Yaskawa INFORM job: A_ROOF_SIDE_0617_2_PAINT_37.JBI

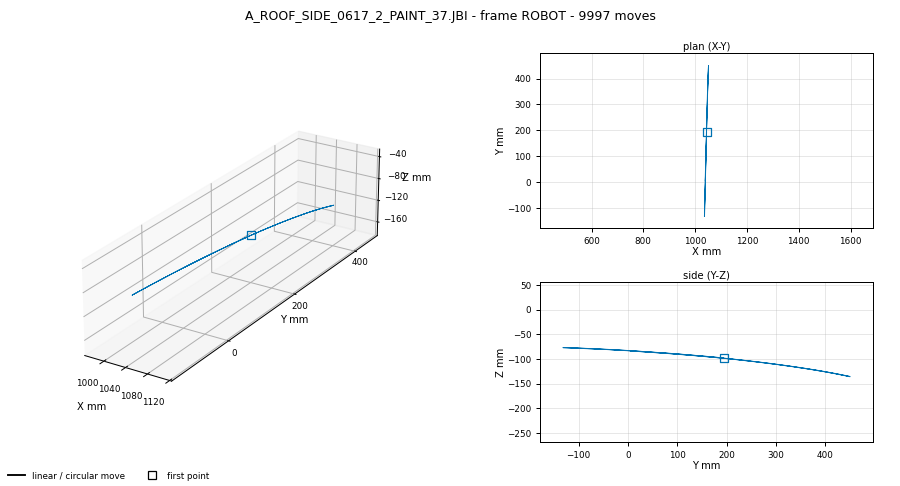
[picture p0: tool path of A_ROOF_SIDE_0617_2_PAINT_37.JBI in frame ROBOT, 9997 of 9997 moves have a stored position in this frame; points joined in program order, loops and branches not executed]
/JOB
//NAME A_ROOF_SIDE_0617_2_PAINT37
//POS
///NPOS 9997,0,0,0,0,0
///TOOL 1
///USER 0
///POSTYPE ROBOT
///RECTAN
///RCONF 1,0,0,0,0,0,0,0,0,0,0,0,0,0,0,0,0,0,0,0,0,0,0,0
C00000=1044.665,193.952,-97.455,170.911,38.372,157.245
C00001=1044.658,193.704,-97.430,170.909,38.370,157.244
C00002=1044.653,193.455,-97.406,170.907,38.368,157.244
C00003=1044.647,193.206,-97.381,170.903,38.367,157.243
C00004=1044.641,192.958,-97.357,170.901,38.365,157.243
C00005=1044.635,192.709,-97.332,170.899,38.364,157.243
C00006=1044.628,192.460,-97.308,170.895,38.362,157.242
C00007=1044.623,192.211,-97.284,170.893,38.360,157.242
C00008=1044.616,191.962,-97.260,170.891,38.359,157.241
C00009=1044.611,191.714,-97.235,170.888,38.357,157.241
C00010=1044.604,191.465,-97.211,170.885,38.355,157.241
C00011=1044.598,191.216,-97.186,170.883,38.353,157.240
C00012=1044.592,190.968,-97.162,170.880,38.352,157.240
C00013=1044.586,190.719,-97.138,170.877,38.350,157.239
C00014=1044.580,190.470,-97.114,170.875,38.348,157.239
C00015=1044.574,190.221,-97.089,170.872,38.347,157.239
C00016=1044.567,189.937,-97.061,170.869,38.345,157.238
C00017=1044.561,189.653,-97.034,170.867,38.342,157.238
C00018=1044.553,189.368,-97.006,170.863,38.341,157.237
C00019=1044.547,189.083,-96.978,170.860,38.339,157.237
C00020=1044.541,188.835,-96.955,170.858,38.337,157.236
C00021=1044.535,188.586,-96.930,170.855,38.336,157.236
C00022=1044.529,188.337,-96.906,170.853,38.334,157.236
C00023=1044.523,188.088,-96.882,170.850,38.332,157.235
C00024=1044.517,187.840,-96.858,170.847,38.330,157.235
C00025=1044.511,187.591,-96.833,170.845,38.329,157.234
C00026=1044.505,187.343,-96.809,170.843,38.327,157.234
C00027=1044.499,187.094,-96.784,170.840,38.325,157.234
C00028=1044.493,186.845,-96.761,170.837,38.323,157.233
C00029=1044.487,186.596,-96.736,170.835,38.322,157.233
C00030=1044.481,186.347,-96.713,170.832,38.320,157.232
C00031=1044.475,186.098,-96.689,170.830,38.319,157.232
C00032=1044.469,185.850,-96.665,170.827,38.317,157.232
C00033=1044.463,185.600,-96.640,170.824,38.315,157.231
C00034=1044.457,185.352,-96.617,170.822,38.313,157.231
C00035=1044.451,185.104,-96.593,170.820,38.312,157.230
C00036=1044.445,184.854,-96.568,170.817,38.310,157.230
C00037=1044.439,184.606,-96.545,170.814,38.308,157.230
C00038=1044.433,184.357,-96.520,170.812,38.307,157.229
C00039=1044.427,184.109,-96.496,170.809,38.305,157.229
C00040=1044.422,183.859,-96.472,170.807,38.304,157.229
C00041=1044.416,183.610,-96.449,170.805,38.302,157.228
C00042=1044.409,183.361,-96.425,170.801,38.300,157.228
C00043=1044.403,183.113,-96.401,170.799,38.299,157.227
C00044=1044.396,182.864,-96.377,170.797,38.297,157.227
C00045=1044.391,182.615,-96.354,170.795,38.296,157.227
C00046=1044.384,182.366,-96.330,170.791,38.294,157.226
C00047=1044.378,182.118,-96.307,170.789,38.293,157.226
C00048=1044.372,181.868,-96.283,170.787,38.291,157.226
C00049=1044.366,181.620,-96.260,170.784,38.290,157.225
C00050=1044.358,181.371,-96.236,170.781,38.289,157.225
C00051=1044.353,181.123,-96.213,170.779,38.287,157.225
C00052=1044.346,180.874,-96.189,170.777,38.286,157.224
C00053=1044.340,180.625,-96.166,170.774,38.284,157.224
C00054=1044.334,180.376,-96.143,170.771,38.283,157.224
C00055=1044.328,180.127,-96.118,170.769,38.281,157.223
C00056=1044.322,179.879,-96.096,170.766,38.279,157.223
C00057=1044.315,179.630,-96.072,170.764,38.278,157.223
C00058=1044.309,179.381,-96.049,170.762,38.276,157.222
C00059=1044.303,179.132,-96.025,170.758,38.275,157.222
C00060=1044.297,178.883,-96.001,170.756,38.274,157.222
C00061=1044.291,178.635,-95.978,170.754,38.272,157.221
C00062=1044.284,178.386,-95.955,170.752,38.271,157.221
C00063=1044.278,178.137,-95.932,170.749,38.270,157.221
C00064=1044.271,177.888,-95.908,170.746,38.268,157.220
C00065=1044.266,177.639,-95.885,170.744,38.266,157.220
C00066=1044.260,177.391,-95.861,170.741,38.265,157.219
C00067=1044.253,177.141,-95.838,170.739,38.263,157.219
C00068=1044.247,176.893,-95.814,170.737,38.262,157.219
C00069=1044.241,176.643,-95.791,170.734,38.260,157.218
C00070=1044.235,176.394,-95.768,170.731,38.259,157.218
C00071=1044.229,176.146,-95.744,170.729,38.257,157.218
C00072=1044.222,175.897,-95.721,170.727,38.256,157.217
C00073=1044.216,175.649,-95.698,170.724,38.255,157.217
C00074=1044.210,175.400,-95.675,170.722,38.253,157.217
C00075=1044.204,175.151,-95.651,170.719,38.252,157.216
C00076=1044.198,174.902,-95.628,170.717,38.251,157.216
C00077=1044.192,174.653,-95.605,170.714,38.249,157.216
C00078=1044.186,174.405,-95.581,170.712,38.248,157.215
C00079=1044.180,174.155,-95.558,170.710,38.246,157.215
C00080=1044.173,173.871,-95.531,170.706,38.244,157.215
C00081=1044.166,173.586,-95.505,170.704,38.242,157.214
C00082=1044.158,173.301,-95.479,170.701,38.241,157.214
C00083=1044.152,173.016,-95.452,170.699,38.239,157.214
C00084=1044.146,172.767,-95.428,170.696,38.238,157.213
C00085=1044.140,172.518,-95.405,170.694,38.237,157.213
C00086=1044.133,172.270,-95.382,170.692,38.235,157.212
C00087=1044.127,172.020,-95.359,170.689,38.234,157.212
C00088=1044.121,171.771,-95.336,170.686,38.232,157.212
C00089=1044.115,171.523,-95.312,170.684,38.231,157.212
C00090=1044.109,171.274,-95.290,170.682,38.229,157.211
C00091=1044.103,171.025,-95.267,170.679,38.228,157.211
C00092=1044.097,170.776,-95.243,170.677,38.226,157.210
C00093=1044.091,170.527,-95.221,170.675,38.224,157.210
C00094=1044.085,170.279,-95.197,170.672,38.223,157.210
C00095=1044.079,170.030,-95.174,170.670,38.221,157.209
C00096=1044.073,169.781,-95.151,170.668,38.220,157.209
C00097=1044.067,169.532,-95.128,170.665,38.219,157.209
C00098=1044.061,169.283,-95.105,170.662,38.217,157.208
C00099=1044.054,169.035,-95.082,170.660,38.216,157.208
C00100=1044.049,168.786,-95.059,170.658,38.214,157.208
C00101=1044.043,168.537,-95.036,170.656,38.213,157.208
C00102=1044.037,168.287,-95.013,170.653,38.212,157.207
C00103=1044.031,168.038,-94.990,170.651,38.210,157.207
C00104=1044.025,167.789,-94.967,170.649,38.209,157.206
C00105=1044.019,167.541,-94.945,170.646,38.207,157.206
C00106=1044.013,167.293,-94.921,170.644,38.206,157.206
C00107=1044.007,167.044,-94.898,170.642,38.205,157.205
C00108=1044.001,166.795,-94.875,170.640,38.203,157.205
C00109=1043.995,166.546,-94.852,170.636,38.202,157.205
C00110=1043.989,166.296,-94.829,170.634,38.200,157.204
C00111=1043.983,166.048,-94.806,170.632,38.199,157.204
C00112=1043.977,165.799,-94.784,170.629,38.197,157.204
C00113=1043.971,165.550,-94.761,170.627,38.196,157.203
C00114=1043.965,165.301,-94.738,170.625,38.194,157.203
C00115=1043.960,165.052,-94.715,170.623,38.193,157.203
C00116=1043.953,164.804,-94.692,170.620,38.191,157.202
C00117=1043.947,164.555,-94.669,170.618,38.190,157.202
C00118=1043.942,164.306,-94.646,170.616,38.188,157.202
C00119=1043.936,164.057,-94.623,170.614,38.187,157.201
C00120=1043.930,163.808,-94.601,170.611,38.185,157.201
C00121=1043.924,163.559,-94.578,170.609,38.184,157.201
C00122=1043.917,163.310,-94.555,170.607,38.182,157.200
C00123=1043.912,163.061,-94.532,170.604,38.181,157.200
C00124=1043.906,162.812,-94.509,170.602,38.179,157.200
C00125=1043.900,162.563,-94.487,170.600,38.178,157.199
C00126=1043.894,162.315,-94.464,170.598,38.177,157.199
C00127=1043.888,162.066,-94.441,170.595,38.175,157.199
C00128=1043.882,161.817,-94.418,170.593,38.174,157.199
C00129=1043.877,161.568,-94.395,170.591,38.172,157.198
C00130=1043.870,161.319,-94.373,170.589,38.171,157.198
C00131=1043.865,161.070,-94.350,170.586,38.170,157.197
C00132=1043.859,160.821,-94.327,170.584,38.168,157.197
C00133=1043.853,160.572,-94.304,170.582,38.167,157.197
C00134=1043.847,160.323,-94.282,170.580,38.165,157.197
C00135=1043.841,160.074,-94.259,170.577,38.164,157.196
C00136=1043.835,159.825,-94.237,170.575,38.162,157.196
C00137=1043.829,159.576,-94.214,170.573,38.161,157.196
C00138=1043.823,159.328,-94.192,170.571,38.160,157.195
C00139=1043.817,159.079,-94.171,170.568,38.158,157.195
C00140=1043.811,158.830,-94.148,170.565,38.157,157.195
C00141=1043.804,158.581,-94.125,170.563,38.156,157.194
C00142=1043.799,158.332,-94.102,170.561,38.155,157.194
C00143=1043.792,158.083,-94.081,170.558,38.153,157.194
C00144=1043.785,157.798,-94.055,170.556,38.152,157.193
C00145=1043.778,157.513,-94.030,170.554,38.150,157.193
C00146=1043.771,157.228,-94.004,170.550,38.149,157.193
C00147=1043.764,156.941,-93.978,170.548,38.147,157.192
C00148=1043.758,156.693,-93.955,170.546,38.146,157.192
C00149=1043.752,156.444,-93.934,170.544,38.145,157.192
C00150=1043.746,156.195,-93.911,170.541,38.143,157.191
C00151=1043.740,155.946,-93.889,170.539,38.142,157.191
C00152=1043.733,155.697,-93.867,170.537,38.141,157.191
C00153=1043.728,155.448,-93.844,170.535,38.140,157.191
C00154=1043.722,155.199,-93.822,170.532,38.138,157.190
C00155=1043.715,154.950,-93.800,170.530,38.137,157.190
C00156=1043.710,154.701,-93.778,170.528,38.136,157.190
C00157=1043.703,154.452,-93.755,170.526,38.135,157.189
C00158=1043.698,154.204,-93.734,170.523,38.133,157.189
C00159=1043.692,153.955,-93.711,170.521,38.132,157.189
C00160=1043.686,153.706,-93.689,170.519,38.130,157.189
C00161=1043.679,153.457,-93.667,170.517,38.129,157.188
C00162=1043.673,153.208,-93.645,170.515,38.128,157.188
C00163=1043.667,152.959,-93.622,170.512,38.126,157.188
C00164=1043.661,152.710,-93.601,170.510,38.125,157.187
C00165=1043.655,152.461,-93.578,170.508,38.124,157.187
C00166=1043.649,152.212,-93.557,170.506,38.123,157.187
C00167=1043.642,151.963,-93.534,170.503,38.122,157.187
C00168=1043.637,151.714,-93.512,170.501,38.121,157.186
C00169=1043.631,151.465,-93.491,170.499,38.119,157.186
C00170=1043.624,151.216,-93.468,170.497,38.118,157.186
C00171=1043.618,150.967,-93.447,170.494,38.116,157.185
C00172=1043.611,150.718,-93.424,170.492,38.115,157.185
C00173=1043.607,150.469,-93.402,170.490,38.114,157.185
C00174=1043.600,150.220,-93.381,170.488,38.112,157.184
C00175=1043.594,149.972,-93.358,170.485,38.111,157.184
C00176=1043.588,149.722,-93.337,170.483,38.110,157.184
C00177=1043.582,149.473,-93.315,170.481,38.109,157.184
C00178=1043.576,149.224,-93.292,170.479,38.108,157.183
C00179=1043.570,148.975,-93.271,170.478,38.107,157.183
C00180=1043.564,148.726,-93.249,170.475,38.105,157.183
C00181=1043.558,148.478,-93.227,170.473,38.104,157.182
C00182=1043.552,148.229,-93.205,170.471,38.102,157.182
C00183=1043.545,147.980,-93.184,170.469,38.101,157.182
C00184=1043.539,147.731,-93.161,170.466,38.100,157.182
C00185=1043.533,147.482,-93.140,170.464,38.099,157.181
C00186=1043.527,147.232,-93.117,170.462,38.098,157.181
C00187=1043.521,146.983,-93.096,170.460,38.097,157.181
C00188=1043.515,146.734,-93.074,170.457,38.095,157.180
C00189=1043.509,146.486,-93.052,170.455,38.094,157.180
C00190=1043.503,146.237,-93.031,170.453,38.092,157.180
C00191=1043.496,145.988,-93.010,170.451,38.091,157.180
C00192=1043.490,145.739,-92.988,170.448,38.090,157.179
C00193=1043.484,145.489,-92.966,170.446,38.089,157.179
C00194=1043.478,145.240,-92.945,170.444,38.088,157.179
C00195=1043.472,144.992,-92.923,170.442,38.087,157.178
C00196=1043.466,144.743,-92.901,170.440,38.086,157.178
C00197=1043.459,144.494,-92.879,170.437,38.084,157.178
C00198=1043.453,144.245,-92.858,170.435,38.083,157.178
C00199=1043.447,143.996,-92.836,170.433,38.082,157.177
C00200=1043.441,143.746,-92.814,170.432,38.081,157.177
C00201=1043.435,143.498,-92.793,170.430,38.080,157.177
C00202=1043.429,143.249,-92.772,170.427,38.078,157.177
C00203=1043.423,142.999,-92.750,170.425,38.077,157.176
C00204=1043.417,142.751,-92.728,170.423,38.076,157.176
C00205=1043.410,142.502,-92.706,170.421,38.074,157.176
C00206=1043.405,142.253,-92.685,170.418,38.073,157.175
C00207=1043.399,142.004,-92.663,170.416,38.072,157.175
C00208=1043.391,141.718,-92.639,170.414,38.071,157.175
C00209=1043.385,141.433,-92.614,170.412,38.070,157.175
C00210=1043.378,141.146,-92.589,170.408,38.068,157.174
C00211=1043.370,140.862,-92.565,170.406,38.067,157.174
C00212=1043.364,140.612,-92.543,170.404,38.066,157.174
C00213=1043.358,140.363,-92.522,170.402,38.064,157.173
C00214=1043.352,140.115,-92.501,170.401,38.063,157.173
C00215=1043.346,139.865,-92.479,170.398,38.062,157.173
C00216=1043.340,139.616,-92.457,170.396,38.060,157.173
C00217=1043.334,139.367,-92.436,170.394,38.059,157.172
C00218=1043.328,139.119,-92.414,170.392,38.058,157.172
C00219=1043.321,138.870,-92.393,170.389,38.057,157.172
C00220=1043.315,138.620,-92.372,170.387,38.056,157.171
C00221=1043.309,138.371,-92.351,170.385,38.054,157.171
C00222=1043.304,138.122,-92.329,170.383,38.053,157.171
C00223=1043.298,137.873,-92.308,170.381,38.052,157.171
C00224=1043.291,137.624,-92.287,170.378,38.051,157.170
C00225=1043.285,137.376,-92.266,170.377,38.050,157.170
C00226=1043.279,137.126,-92.244,170.375,38.049,157.170
C00227=1043.273,136.877,-92.222,170.373,38.047,157.170
C00228=1043.266,136.628,-92.202,170.371,38.047,157.169
C00229=1043.261,136.379,-92.181,170.368,38.046,157.169
C00230=1043.255,136.130,-92.159,170.366,38.045,157.169
C00231=1043.248,135.881,-92.138,170.364,38.043,157.169
C00232=1043.242,135.632,-92.117,170.362,38.042,157.168
C00233=1043.236,135.383,-92.096,170.359,38.041,157.168
C00234=1043.229,135.134,-92.075,170.357,38.040,157.168
C00235=1043.224,134.885,-92.053,170.356,38.039,157.168
C00236=1043.218,134.636,-92.032,170.354,38.037,157.167
C00237=1043.211,134.387,-92.012,170.352,38.036,157.167
C00238=1043.206,134.138,-91.990,170.349,38.035,157.167
C00239=1043.199,133.889,-91.969,170.347,38.034,157.167
C00240=1043.192,133.640,-91.948,170.345,38.033,157.166
C00241=1043.187,133.391,-91.927,170.343,38.032,157.166
C00242=1043.181,133.142,-91.905,170.341,38.030,157.166
C00243=1043.174,132.893,-91.884,170.338,38.029,157.165
C00244=1043.169,132.644,-91.864,170.337,38.028,157.165
C00245=1043.163,132.394,-91.842,170.335,38.027,157.165
C00246=1043.156,132.146,-91.821,170.333,38.026,157.165
C00247=1043.151,131.896,-91.801,170.330,38.025,157.164
C00248=1043.144,131.647,-91.779,170.328,38.023,157.164
C00249=1043.138,131.399,-91.758,170.326,38.022,157.164
C00250=1043.132,131.149,-91.737,170.324,38.021,157.164
C00251=1043.125,130.900,-91.716,170.323,38.020,157.163
C00252=1043.120,130.651,-91.696,170.321,38.019,157.163
C00253=1043.113,130.402,-91.675,170.318,38.018,157.163
C00254=1043.107,130.152,-91.654,170.316,38.017,157.163
C00255=1043.101,129.904,-91.633,170.314,38.016,157.162
C00256=1043.094,129.655,-91.613,170.312,38.015,157.162
C00257=1043.088,129.405,-91.591,170.309,38.013,157.162
C00258=1043.082,129.157,-91.571,170.307,38.013,157.162
C00259=1043.075,128.908,-91.550,170.305,38.012,157.161
C00260=1043.070,128.659,-91.530,170.304,38.011,157.161
C00261=1043.063,128.410,-91.509,170.302,38.009,157.161
C00262=1043.057,128.160,-91.488,170.300,38.008,157.161
C00263=1043.051,127.912,-91.467,170.297,38.008,157.161
C00264=1043.044,127.662,-91.447,170.295,38.006,157.160
C00265=1043.039,127.414,-91.425,170.293,38.005,157.160
C00266=1043.032,127.164,-91.405,170.291,38.004,157.160
C00267=1043.025,126.915,-91.384,170.289,38.003,157.159
C00268=1043.020,126.666,-91.363,170.287,38.002,157.159
C00269=1043.013,126.417,-91.342,170.285,38.001,157.159
C00270=1043.007,126.168,-91.322,170.283,38.000,157.159
C00271=1043.001,125.919,-91.302,170.281,37.999,157.159
C00272=1042.994,125.633,-91.278,170.279,37.998,157.158
C00273=1042.987,125.347,-91.254,170.276,37.996,157.158
C00274=1042.980,125.062,-91.230,170.274,37.995,157.158
C00275=1042.972,124.775,-91.207,170.271,37.994,157.157
C00276=1042.966,124.527,-91.186,170.270,37.993,157.157
C00277=1042.960,124.277,-91.165,170.268,37.992,157.157
C00278=1042.954,124.028,-91.145,170.265,37.991,157.157
C00279=1042.947,123.779,-91.124,170.263,37.989,157.156
C00280=1042.942,123.530,-91.104,170.261,37.988,157.156
C00281=1042.936,123.281,-91.083,170.259,37.987,157.156
C00282=1042.929,123.032,-91.063,170.257,37.987,157.156
C00283=1042.923,122.783,-91.042,170.255,37.985,157.156
C00284=1042.917,122.534,-91.022,170.253,37.984,157.155
C00285=1042.911,122.285,-91.001,170.251,37.983,157.155
C00286=1042.905,122.036,-90.980,170.249,37.982,157.155
C00287=1042.899,121.786,-90.960,170.247,37.981,157.154
C00288=1042.893,121.538,-90.940,170.244,37.979,157.154
C00289=1042.886,121.289,-90.919,170.243,37.979,157.154
C00290=1042.881,121.039,-90.898,170.241,37.978,157.154
C00291=1042.874,120.790,-90.878,170.239,37.977,157.154
C00292=1042.868,120.541,-90.858,170.237,37.975,157.153
C00293=1042.862,120.293,-90.837,170.234,37.974,157.153
C00294=1042.856,120.043,-90.816,170.233,37.973,157.153
C00295=1042.850,119.794,-90.797,170.231,37.972,157.152
C00296=1042.844,119.544,-90.776,170.229,37.971,157.152
C00297=1042.838,119.296,-90.756,170.227,37.970,157.152
C00298=1042.831,119.047,-90.735,170.224,37.969,157.152
C00299=1042.825,118.798,-90.715,170.222,37.968,157.152
C00300=1042.820,118.549,-90.694,170.221,37.966,157.151
C00301=1042.813,118.299,-90.674,170.219,37.965,157.151
C00302=1042.807,118.051,-90.654,170.217,37.964,157.151
C00303=1042.801,117.801,-90.633,170.214,37.963,157.150
C00304=1042.795,117.553,-90.612,170.212,37.962,157.150
C00305=1042.788,117.303,-90.592,170.211,37.961,157.150
C00306=1042.782,117.054,-90.572,170.209,37.960,157.150
C00307=1042.777,116.805,-90.551,170.207,37.959,157.150
C00308=1042.771,116.556,-90.531,170.204,37.958,157.149
C00309=1042.765,116.307,-90.511,170.202,37.956,157.149
C00310=1042.759,116.058,-90.491,170.201,37.955,157.149
C00311=1042.753,115.808,-90.470,170.199,37.954,157.149
C00312=1042.747,115.559,-90.450,170.197,37.953,157.148
C00313=1042.740,115.311,-90.430,170.195,37.952,157.148
C00314=1042.735,115.061,-90.409,170.192,37.951,157.148
C00315=1042.729,114.812,-90.389,170.191,37.950,157.148
C00316=1042.723,114.564,-90.369,170.189,37.949,157.147
C00317=1042.716,114.314,-90.348,170.187,37.948,157.147
C00318=1042.711,114.065,-90.328,170.184,37.946,157.147
C00319=1042.705,113.816,-90.308,170.183,37.945,157.147
C00320=1042.698,113.567,-90.288,170.181,37.944,157.146
C00321=1042.692,113.318,-90.268,170.179,37.943,157.146
C00322=1042.686,113.068,-90.247,170.177,37.942,157.146
C00323=1042.680,112.820,-90.227,170.175,37.941,157.146
C00324=1042.674,112.571,-90.207,170.173,37.940,157.145
C00325=1042.667,112.321,-90.188,170.171,37.939,157.145
C00326=1042.661,112.072,-90.168,170.169,37.938,157.145
C00327=1042.655,111.823,-90.148,170.167,37.937,157.145
C00328=1042.649,111.573,-90.128,170.165,37.936,157.144
C00329=1042.643,111.325,-90.108,170.163,37.935,157.144
C00330=1042.637,111.076,-90.088,170.161,37.934,157.144
C00331=1042.630,110.826,-90.067,170.159,37.933,157.144
C00332=1042.624,110.577,-90.047,170.157,37.932,157.144
C00333=1042.618,110.329,-90.027,170.155,37.930,157.143
C00334=1042.612,110.079,-90.008,170.154,37.930,157.143
C00335=1042.606,109.830,-89.988,170.151,37.929,157.143
C00336=1042.599,109.544,-89.965,170.149,37.928,157.143
C00337=1042.591,109.257,-89.942,170.147,37.926,157.142
C00338=1042.584,108.971,-89.919,170.144,37.925,157.142
C00339=1042.577,108.686,-89.897,170.142,37.924,157.142
C00340=1042.571,108.437,-89.877,170.140,37.923,157.142
C00341=1042.564,108.187,-89.857,170.138,37.922,157.141
C00342=1042.558,107.938,-89.837,170.136,37.921,157.141
C00343=1042.553,107.689,-89.817,170.134,37.920,157.141
C00344=1042.546,107.441,-89.798,170.132,37.919,157.141
C00345=1042.539,107.191,-89.778,170.130,37.918,157.140
C00346=1042.533,106.942,-89.758,170.128,37.917,157.140
C00347=1042.528,106.693,-89.739,170.126,37.916,157.140
C00348=1042.521,106.443,-89.718,170.124,37.915,157.140
C00349=1042.515,106.194,-89.698,170.122,37.914,157.140
C00350=1042.509,105.945,-89.680,170.121,37.913,157.139
C00351=1042.503,105.696,-89.660,170.118,37.912,157.139
C00352=1042.496,105.447,-89.639,170.116,37.911,157.139
C00353=1042.490,105.198,-89.620,170.114,37.910,157.139
C00354=1042.484,104.949,-89.600,170.113,37.909,157.139
C00355=1042.478,104.700,-89.580,170.111,37.908,157.138
C00356=1042.471,104.450,-89.561,170.109,37.907,157.138
C00357=1042.465,104.201,-89.541,170.106,37.906,157.138
C00358=1042.459,103.952,-89.521,170.104,37.905,157.138
C00359=1042.454,103.703,-89.502,170.103,37.904,157.137
C00360=1042.447,103.454,-89.482,170.101,37.903,157.137
C00361=1042.441,103.204,-89.463,170.099,37.902,157.137
C00362=1042.435,102.956,-89.443,170.096,37.901,157.137
C00363=1042.429,102.707,-89.423,170.095,37.900,157.136
C00364=1042.423,102.457,-89.404,170.093,37.899,157.136
C00365=1042.416,102.208,-89.383,170.091,37.897,157.136
C00366=1042.411,101.958,-89.364,170.089,37.897,157.136
C00367=1042.404,101.710,-89.345,170.087,37.896,157.135
C00368=1042.398,101.461,-89.325,170.085,37.894,157.135
C00369=1042.392,101.212,-89.306,170.083,37.893,157.135
C00370=1042.386,100.962,-89.285,170.081,37.893,157.135
C00371=1042.380,100.713,-89.266,170.079,37.892,157.135
C00372=1042.373,100.464,-89.247,170.078,37.890,157.134
C00373=1042.368,100.215,-89.227,170.076,37.890,157.134
C00374=1042.362,99.966,-89.208,170.073,37.889,157.134
C00375=1042.355,99.716,-89.189,170.071,37.887,157.134
C00376=1042.349,99.467,-89.169,170.070,37.887,157.134
C00377=1042.342,99.218,-89.150,170.068,37.886,157.133
C00378=1042.337,98.969,-89.131,170.066,37.884,157.133
C00379=1042.330,98.720,-89.111,170.063,37.884,157.133
C00380=1042.323,98.470,-89.092,170.061,37.883,157.133
C00381=1042.317,98.222,-89.072,170.060,37.882,157.132
C00382=1042.311,97.972,-89.053,170.058,37.881,157.132
C00383=1042.305,97.723,-89.034,170.056,37.880,157.132
C00384=1042.299,97.474,-89.014,170.054,37.879,157.132
C00385=1042.292,97.224,-88.995,170.051,37.878,157.132
C00386=1042.286,96.976,-88.976,170.050,37.877,157.131
C00387=1042.280,96.726,-88.956,170.048,37.876,157.131
C00388=1042.274,96.477,-88.938,170.046,37.875,157.131
C00389=1042.268,96.228,-88.918,170.044,37.874,157.131
C00390=1042.261,95.979,-88.899,170.043,37.873,157.130
C00391=1042.255,95.730,-88.880,170.040,37.872,157.130
C00392=1042.248,95.480,-88.860,170.038,37.871,157.130
C00393=1042.242,95.231,-88.841,170.036,37.870,157.130
C00394=1042.236,94.982,-88.822,170.035,37.869,157.130
C00395=1042.230,94.732,-88.803,170.033,37.868,157.129
C00396=1042.224,94.484,-88.784,170.031,37.867,157.129
C00397=1042.218,94.235,-88.764,170.028,37.866,157.129
C00398=1042.212,93.985,-88.745,170.026,37.866,157.129
C00399=1042.205,93.737,-88.726,170.025,37.864,157.129
C00400=1042.198,93.450,-88.704,170.023,37.863,157.128
C00401=1042.191,93.165,-88.682,170.021,37.862,157.128
C00402=1042.184,92.878,-88.660,170.018,37.861,157.128
C00403=1042.177,92.592,-88.638,170.016,37.860,157.127
C00404=1042.171,92.343,-88.618,170.014,37.859,157.127
C00405=1042.165,92.094,-88.599,170.012,37.858,157.127
C00406=1042.158,91.845,-88.581,170.010,37.857,157.127
C00407=1042.153,91.595,-88.561,170.009,37.856,157.127
C00408=1042.146,91.346,-88.543,170.006,37.855,157.126
C00409=1042.140,91.097,-88.523,170.004,37.854,157.126
C00410=1042.134,90.848,-88.504,170.002,37.853,157.126
C00411=1042.128,90.599,-88.485,170.001,37.852,157.126
C00412=1042.122,90.350,-88.466,169.999,37.851,157.126
C00413=1042.116,90.100,-88.447,169.997,37.850,157.125
C00414=1042.109,89.850,-88.428,169.994,37.849,157.125
C00415=1042.103,89.601,-88.409,169.993,37.848,157.125
C00416=1042.096,89.353,-88.390,169.991,37.847,157.125
C00417=1042.090,89.103,-88.371,169.989,37.846,157.124
C00418=1042.084,88.854,-88.352,169.987,37.845,157.124
C00419=1042.077,88.605,-88.333,169.985,37.844,157.124
C00420=1042.071,88.356,-88.315,169.984,37.844,157.124
C00421=1042.065,88.106,-88.296,169.981,37.842,157.124
C00422=1042.059,87.857,-88.277,169.979,37.842,157.124
C00423=1042.052,87.608,-88.258,169.977,37.841,157.123
C00424=1042.046,87.359,-88.240,169.976,37.840,157.123
C00425=1042.040,87.110,-88.220,169.974,37.839,157.123
C00426=1042.034,86.861,-88.202,169.972,37.838,157.123
C00427=1042.027,86.611,-88.183,169.969,37.837,157.122
C00428=1042.021,86.362,-88.164,169.967,37.836,157.122
C00429=1042.015,86.113,-88.146,169.966,37.835,157.122
C00430=1042.009,85.864,-88.126,169.964,37.834,157.122
C00431=1042.003,85.615,-88.108,169.962,37.834,157.122
C00432=1041.996,85.365,-88.089,169.960,37.832,157.121
C00433=1041.990,85.116,-88.071,169.958,37.832,157.121
C00434=1041.984,84.867,-88.051,169.956,37.831,157.121
C00435=1041.978,84.618,-88.033,169.954,37.829,157.121
C00436=1041.971,84.369,-88.014,169.952,37.829,157.121
C00437=1041.965,84.120,-87.995,169.951,37.828,157.120
C00438=1041.958,83.870,-87.977,169.949,37.827,157.120
C00439=1041.953,83.620,-87.958,169.946,37.826,157.120
C00440=1041.946,83.371,-87.940,169.944,37.825,157.120
C00441=1041.940,83.122,-87.921,169.943,37.824,157.120
C00442=1041.934,82.873,-87.902,169.941,37.823,157.119
C00443=1041.927,82.624,-87.884,169.939,37.822,157.119
C00444=1041.922,82.374,-87.864,169.937,37.821,157.119
C00445=1041.915,82.125,-87.846,169.936,37.820,157.119
C00446=1041.909,81.876,-87.827,169.933,37.819,157.119
C00447=1041.902,81.627,-87.808,169.931,37.818,157.118
C00448=1041.896,81.377,-87.790,169.929,37.818,157.118
C00449=1041.890,81.128,-87.771,169.928,37.816,157.118
C00450=1041.884,80.879,-87.753,169.926,37.816,157.118
C00451=1041.878,80.630,-87.734,169.924,37.815,157.118
C00452=1041.872,80.381,-87.716,169.921,37.813,157.117
C00453=1041.866,80.132,-87.698,169.920,37.813,157.117
C00454=1041.860,79.882,-87.678,169.918,37.812,157.117
C00455=1041.854,79.633,-87.660,169.916,37.811,157.117
C00456=1041.847,79.384,-87.641,169.914,37.810,157.116
C00457=1041.841,79.135,-87.623,169.913,37.809,157.116
C00458=1041.835,78.885,-87.605,169.910,37.808,157.116
C00459=1041.828,78.636,-87.586,169.908,37.807,157.116
C00460=1041.822,78.386,-87.567,169.906,37.806,157.116
C00461=1041.816,78.137,-87.548,169.905,37.805,157.115
C00462=1041.810,77.888,-87.530,169.903,37.804,157.115
C00463=1041.804,77.639,-87.512,169.901,37.803,157.115
C00464=1041.796,77.353,-87.491,169.898,37.802,157.115
C00465=1041.789,77.067,-87.469,169.896,37.801,157.115
C00466=1041.782,76.781,-87.449,169.894,37.800,157.114
C00467=1041.775,76.495,-87.428,169.892,37.799,157.114
C00468=1041.769,76.245,-87.409,169.890,37.798,157.114
C00469=1041.762,75.996,-87.390,169.888,37.797,157.114
C00470=1041.756,75.747,-87.372,169.886,37.796,157.113
C00471=1041.750,75.498,-87.354,169.884,37.796,157.113
C00472=1041.744,75.248,-87.336,169.882,37.794,157.113
C00473=1041.738,74.999,-87.317,169.880,37.794,157.113
C00474=1041.730,74.750,-87.299,169.879,37.793,157.113
C00475=1041.724,74.501,-87.281,169.877,37.792,157.113
C00476=1041.718,74.252,-87.263,169.875,37.791,157.112
C00477=1041.712,74.002,-87.245,169.872,37.790,157.112
C00478=1041.706,73.753,-87.227,169.871,37.789,157.112
C00479=1041.700,73.504,-87.208,169.869,37.788,157.112
C00480=1041.693,73.255,-87.190,169.867,37.787,157.112
C00481=1041.687,73.005,-87.171,169.865,37.787,157.111
C00482=1041.681,72.756,-87.153,169.863,37.785,157.111
C00483=1041.674,72.507,-87.135,169.861,37.785,157.111
C00484=1041.669,72.258,-87.117,169.859,37.784,157.111
C00485=1041.662,72.008,-87.099,169.857,37.783,157.111
C00486=1041.656,71.759,-87.081,169.855,37.782,157.110
C00487=1041.649,71.510,-87.063,169.854,37.781,157.110
C00488=1041.643,71.260,-87.045,169.852,37.780,157.110
C00489=1041.637,71.011,-87.026,169.850,37.779,157.110
C00490=1041.631,70.762,-87.008,169.847,37.778,157.110
C00491=1041.625,70.513,-86.990,169.846,37.778,157.109
C00492=1041.619,70.263,-86.972,169.844,37.776,157.109
C00493=1041.612,70.014,-86.953,169.842,37.775,157.109
C00494=1041.606,69.765,-86.936,169.840,37.775,157.109
C00495=1041.600,69.515,-86.918,169.839,37.773,157.109
C00496=1041.593,69.266,-86.900,169.836,37.773,157.108
C00497=1041.587,69.017,-86.882,169.834,37.772,157.108
C00498=1041.581,68.768,-86.863,169.832,37.771,157.108
C00499=1041.575,68.519,-86.846,169.831,37.771,157.108
C00500=1041.568,68.269,-86.828,169.829,37.769,157.108
C00501=1041.562,68.020,-86.810,169.827,37.769,157.107
C00502=1041.556,67.770,-86.792,169.825,37.768,157.107
C00503=1041.549,67.522,-86.774,169.822,37.767,157.107
C00504=1041.543,67.272,-86.756,169.821,37.766,157.107
C00505=1041.537,67.023,-86.738,169.819,37.765,157.107
C00506=1041.531,66.773,-86.719,169.817,37.764,157.106
C00507=1041.524,66.524,-86.702,169.815,37.763,157.106
C00508=1041.518,66.275,-86.685,169.814,37.762,157.106
C00509=1041.512,66.025,-86.667,169.812,37.762,157.106
C00510=1041.505,65.776,-86.649,169.809,37.760,157.106
C00511=1041.499,65.527,-86.631,169.807,37.760,157.106
C00512=1041.493,65.278,-86.613,169.805,37.759,157.105
C00513=1041.486,65.029,-86.595,169.804,37.758,157.105
C00514=1041.480,64.779,-86.577,169.802,37.757,157.105
C00515=1041.475,64.530,-86.559,169.800,37.756,157.105
C00516=1041.468,64.281,-86.542,169.798,37.756,157.105
C00517=1041.461,64.032,-86.523,169.796,37.754,157.104
C00518=1041.455,63.782,-86.506,169.794,37.754,157.104
C00519=1041.449,63.533,-86.489,169.792,37.753,157.104
C00520=1041.443,63.283,-86.471,169.790,37.752,157.104
C00521=1041.436,63.034,-86.453,169.788,37.752,157.104
C00522=1041.429,62.784,-86.436,169.787,37.750,157.103
C00523=1041.423,62.536,-86.418,169.785,37.750,157.103
C00524=1041.416,62.287,-86.400,169.782,37.749,157.103
C00525=1041.410,62.037,-86.382,169.780,37.748,157.103
C00526=1041.403,61.787,-86.365,169.778,37.747,157.103
C00527=1041.397,61.539,-86.348,169.777,37.747,157.103
C00528=1041.390,61.252,-86.328,169.775,37.746,157.102
C00529=1041.382,60.965,-86.307,169.772,37.745,157.102
C00530=1041.375,60.679,-86.288,169.770,37.744,157.102
C00531=1041.367,60.393,-86.267,169.767,37.743,157.102
C00532=1041.362,60.144,-86.250,169.766,37.742,157.102
C00533=1041.355,59.894,-86.232,169.764,37.742,157.101
C00534=1041.348,59.646,-86.214,169.762,37.741,157.101
C00535=1041.342,59.397,-86.197,169.760,37.740,157.101
C00536=1041.336,59.147,-86.179,169.758,37.739,157.101
C00537=1041.329,58.897,-86.161,169.757,37.739,157.101
C00538=1041.323,58.649,-86.144,169.754,37.737,157.101
C00539=1041.316,58.399,-86.127,169.752,37.737,157.100
C00540=1041.310,58.149,-86.109,169.750,37.736,157.100
C00541=1041.304,57.901,-86.092,169.748,37.735,157.100
C00542=1041.298,57.651,-86.074,169.747,37.734,157.100
C00543=1041.291,57.402,-86.057,169.745,37.733,157.100
C00544=1041.285,57.153,-86.040,169.743,37.733,157.100
C00545=1041.279,56.903,-86.022,169.741,37.732,157.099
C00546=1041.272,56.654,-86.005,169.738,37.731,157.099
C00547=1041.265,56.405,-85.988,169.737,37.730,157.099
C00548=1041.259,56.155,-85.970,169.735,37.730,157.099
C00549=1041.253,55.906,-85.952,169.733,37.728,157.099
C00550=1041.247,55.656,-85.936,169.731,37.728,157.098
C00551=1041.240,55.407,-85.918,169.729,37.727,157.098
C00552=1041.234,55.158,-85.901,169.728,37.726,157.098
C00553=1041.228,54.908,-85.883,169.725,37.726,157.098
C00554=1041.221,54.659,-85.866,169.723,37.724,157.098
C00555=1041.215,54.410,-85.849,169.721,37.724,157.098
C00556=1041.209,54.160,-85.831,169.719,37.723,157.097
C00557=1041.203,53.912,-85.814,169.718,37.722,157.097
C00558=1041.196,53.662,-85.796,169.716,37.721,157.097
C00559=1041.190,53.413,-85.779,169.714,37.720,157.097
C00560=1041.183,53.164,-85.762,169.711,37.720,157.097
C00561=1041.178,52.913,-85.745,169.709,37.719,157.096
C00562=1041.171,52.665,-85.728,169.708,37.718,157.096
C00563=1041.164,52.415,-85.710,169.706,37.717,157.096
C00564=1041.159,52.166,-85.693,169.704,37.717,157.096
C00565=1041.152,51.917,-85.675,169.702,37.715,157.096
C00566=1041.146,51.668,-85.658,169.701,37.715,157.096
C00567=1041.140,51.418,-85.641,169.698,37.714,157.095
C00568=1041.134,51.169,-85.624,169.696,37.713,157.095
C00569=1041.127,50.919,-85.607,169.694,37.712,157.095
C00570=1041.121,50.670,-85.589,169.692,37.711,157.095
C00571=1041.114,50.421,-85.572,169.691,37.711,157.095
C00572=1041.108,50.171,-85.555,169.689,37.709,157.094
C00573=1041.102,49.922,-85.538,169.687,37.709,157.094
C00574=1041.096,49.672,-85.521,169.685,37.708,157.094
C00575=1041.089,49.424,-85.504,169.682,37.707,157.094
C00576=1041.083,49.174,-85.486,169.681,37.706,157.094
C00577=1041.077,48.925,-85.469,169.679,37.705,157.094
C00578=1041.071,48.676,-85.452,169.677,37.705,157.093
C00579=1041.065,48.426,-85.434,169.675,37.703,157.093
C00580=1041.059,48.177,-85.418,169.673,37.703,157.093
C00581=1041.052,47.927,-85.401,169.672,37.702,157.093
C00582=1041.047,47.678,-85.383,169.669,37.701,157.093
C00583=1041.040,47.429,-85.366,169.667,37.701,157.092
C00584=1041.034,47.180,-85.350,169.665,37.699,157.092
C00585=1041.028,46.930,-85.332,169.664,37.699,157.092
C00586=1041.021,46.681,-85.315,169.662,37.697,157.092
C00587=1041.015,46.431,-85.298,169.660,37.697,157.092
C00588=1041.009,46.182,-85.281,169.658,37.696,157.091
C00589=1041.003,45.933,-85.264,169.655,37.695,157.091
C00590=1040.996,45.683,-85.247,169.654,37.695,157.091
C00591=1040.991,45.434,-85.229,169.652,37.693,157.091
C00592=1040.985,45.188,-85.212,169.650,37.693,157.091
C00593=1040.979,44.943,-85.196,169.648,37.692,157.091
C00594=1040.972,44.698,-85.179,169.647,37.691,157.090
C00595=1040.967,44.452,-85.163,169.645,37.690,157.090
C00596=1040.960,44.206,-85.146,169.642,37.689,157.090
C00597=1040.955,43.961,-85.129,169.640,37.689,157.090
C00598=1040.948,43.716,-85.112,169.639,37.687,157.090
C00599=1040.942,43.471,-85.096,169.637,37.687,157.089
C00600=1040.936,43.221,-85.079,169.635,37.686,157.089
C00601=1040.929,42.972,-85.061,169.633,37.685,157.089
C00602=1040.924,42.722,-85.045,169.631,37.684,157.089
C00603=1040.917,42.473,-85.028,169.629,37.683,157.089
C00604=1040.911,42.224,-85.012,169.627,37.683,157.089
C00605=1040.904,41.974,-84.994,169.625,37.682,157.088
C00606=1040.898,41.725,-84.978,169.623,37.681,157.088
C00607=1040.892,41.476,-84.961,169.621,37.680,157.088
C00608=1040.885,41.226,-84.944,169.619,37.680,157.088
C00609=1040.879,40.977,-84.927,169.618,37.678,157.088
C00610=1040.872,40.727,-84.911,169.616,37.678,157.088
C00611=1040.866,40.479,-84.894,169.613,37.677,157.087
C00612=1040.860,40.229,-84.878,169.611,37.676,157.087
C00613=1040.854,39.979,-84.861,169.609,37.675,157.087
C00614=1040.847,39.730,-84.844,169.607,37.675,157.087
C00615=1040.841,39.481,-84.828,169.606,37.674,157.087
C00616=1040.835,39.231,-84.810,169.604,37.673,157.087
C00617=1040.829,38.982,-84.794,169.602,37.672,157.086
C00618=1040.822,38.733,-84.776,169.600,37.671,157.086
C00619=1040.816,38.483,-84.760,169.597,37.671,157.086
C00620=1040.811,38.234,-84.744,169.596,37.670,157.086
C00621=1040.804,37.984,-84.726,169.594,37.669,157.086
C00622=1040.798,37.735,-84.710,169.592,37.668,157.085
C00623=1040.792,37.486,-84.694,169.590,37.668,157.085
C00624=1040.785,37.236,-84.676,169.588,37.666,157.085
C00625=1040.778,36.987,-84.661,169.586,37.666,157.085
C00626=1040.772,36.738,-84.645,169.585,37.665,157.085
C00627=1040.765,36.489,-84.627,169.582,37.665,157.085
C00628=1040.759,36.239,-84.611,169.580,37.664,157.085
C00629=1040.753,35.990,-84.595,169.578,37.663,157.084
C00630=1040.747,35.740,-84.578,169.576,37.662,157.084
C00631=1040.740,35.491,-84.562,169.574,37.662,157.084
C00632=1040.734,35.242,-84.545,169.572,37.661,157.084
C00633=1040.727,34.992,-84.529,169.571,37.660,157.084
C00634=1040.721,34.743,-84.513,169.569,37.659,157.084
C00635=1040.715,34.494,-84.496,169.566,37.659,157.083
C00636=1040.707,34.199,-84.476,169.564,37.658,157.083
C00637=1040.700,33.904,-84.457,169.561,37.657,157.083
C00638=1040.693,33.610,-84.437,169.559,37.656,157.083
C00639=1040.685,33.315,-84.418,169.557,37.655,157.083
C00640=1040.679,33.066,-84.403,169.555,37.655,157.082
C00641=1040.672,32.817,-84.385,169.553,37.654,157.082
C00642=1040.666,32.568,-84.369,169.551,37.653,157.082
C00643=1040.660,32.318,-84.353,169.549,37.652,157.082
C00644=1040.653,32.068,-84.336,169.547,37.652,157.082
C00645=1040.647,31.819,-84.321,169.545,37.651,157.082
C00646=1040.641,31.570,-84.304,169.543,37.650,157.081
C00647=1040.635,31.320,-84.288,169.541,37.649,157.081
C00648=1040.628,31.071,-84.271,169.539,37.649,157.081
C00649=1040.621,30.822,-84.255,169.538,37.648,157.081
C00650=1040.615,30.573,-84.239,169.535,37.647,157.081
C00651=1040.609,30.323,-84.222,169.533,37.646,157.081
C00652=1040.603,30.073,-84.206,169.531,37.646,157.081
C00653=1040.597,29.824,-84.190,169.529,37.645,157.080
C00654=1040.590,29.575,-84.174,169.527,37.644,157.080
C00655=1040.584,29.326,-84.158,169.525,37.643,157.080
C00656=1040.576,29.039,-84.139,169.523,37.643,157.080
C00657=1040.570,28.752,-84.119,169.521,37.642,157.080
C00658=1040.562,28.465,-84.102,169.518,37.641,157.079
C00659=1040.555,28.179,-84.083,169.516,37.640,157.079
C00660=1040.549,27.930,-84.067,169.514,37.639,157.079
C00661=1040.542,27.680,-84.051,169.512,37.639,157.079
C00662=1040.536,27.430,-84.034,169.510,37.638,157.079
C00663=1040.530,27.181,-84.018,169.508,37.637,157.079
C00664=1040.523,26.932,-84.002,169.506,37.636,157.078
C00665=1040.517,26.683,-83.986,169.505,37.636,157.078
C00666=1040.511,26.433,-83.970,169.503,37.635,157.078
C00667=1040.504,26.184,-83.954,169.500,37.634,157.078
C00668=1040.498,25.934,-83.938,169.498,37.634,157.078
C00669=1040.491,25.685,-83.922,169.496,37.633,157.078
C00670=1040.485,25.435,-83.906,169.494,37.632,157.078
C00671=1040.478,25.186,-83.890,169.492,37.632,157.077
C00672=1040.473,24.936,-83.874,169.490,37.631,157.077
C00673=1040.467,24.687,-83.858,169.488,37.630,157.077
C00674=1040.460,24.438,-83.842,169.487,37.630,157.077
C00675=1040.454,24.188,-83.826,169.485,37.629,157.077
C00676=1040.447,23.939,-83.810,169.482,37.628,157.077
C00677=1040.441,23.689,-83.794,169.480,37.627,157.076
C00678=1040.434,23.440,-83.778,169.478,37.627,157.076
C00679=1040.428,23.190,-83.762,169.476,37.626,157.076
C00680=1040.422,22.941,-83.747,169.474,37.626,157.076
C00681=1040.416,22.692,-83.731,169.472,37.625,157.076
C00682=1040.408,22.442,-83.715,169.470,37.624,157.076
C00683=1040.402,22.193,-83.698,169.469,37.623,157.076
C00684=1040.397,21.944,-83.682,169.466,37.623,157.075
C00685=1040.390,21.694,-83.667,169.464,37.622,157.075
C00686=1040.384,21.445,-83.651,169.462,37.621,157.075
C00687=1040.377,21.196,-83.635,169.460,37.621,157.075
C00688=1040.372,20.946,-83.619,169.458,37.620,157.075
C00689=1040.365,20.697,-83.604,169.456,37.619,157.075
C00690=1040.359,20.446,-83.587,169.454,37.618,157.075
C00691=1040.352,20.197,-83.572,169.452,37.618,157.074
C00692=1040.346,19.948,-83.555,169.450,37.617,157.074
C00693=1040.340,19.698,-83.540,169.448,37.617,157.074
C00694=1040.334,19.449,-83.524,169.446,37.615,157.074
C00695=1040.327,19.200,-83.509,169.444,37.615,157.074
C00696=1040.320,18.951,-83.493,169.442,37.614,157.074
C00697=1040.315,18.701,-83.477,169.440,37.614,157.073
C00698=1040.308,18.452,-83.462,169.438,37.613,157.073
C00699=1040.302,18.203,-83.445,169.436,37.613,157.073
C00700=1040.295,17.952,-83.430,169.434,37.612,157.073
C00701=1040.288,17.703,-83.414,169.432,37.611,157.073
C00702=1040.282,17.454,-83.398,169.430,37.611,157.073
C00703=1040.276,17.204,-83.383,169.427,37.610,157.073
C00704=1040.270,16.955,-83.367,169.425,37.609,157.072
C00705=1040.264,16.705,-83.352,169.423,37.608,157.072
C00706=1040.257,16.456,-83.336,169.422,37.608,157.072
C00707=1040.251,16.207,-83.320,169.420,37.607,157.072
C00708=1040.245,15.957,-83.305,169.418,37.607,157.072
C00709=1040.238,15.708,-83.290,169.416,37.606,157.072
C00710=1040.232,15.458,-83.274,169.414,37.605,157.072
C00711=1040.226,15.209,-83.258,169.411,37.604,157.071
C00712=1040.220,14.960,-83.242,169.409,37.604,157.071
C00713=1040.213,14.710,-83.227,169.407,37.603,157.071
C00714=1040.207,14.461,-83.211,169.405,37.603,157.071
C00715=1040.201,14.211,-83.196,169.403,37.602,157.071
C00716=1040.194,13.962,-83.180,169.401,37.601,157.071
C00717=1040.188,13.712,-83.165,169.399,37.601,157.071
C00718=1040.181,13.463,-83.150,169.397,37.600,157.070
C00719=1040.175,13.214,-83.135,169.395,37.600,157.070
C00720=1040.167,12.929,-83.117,169.393,37.599,157.070
C00721=1040.160,12.643,-83.099,169.390,37.598,157.070
C00722=1040.153,12.358,-83.081,169.388,37.598,157.070
C00723=1040.146,12.072,-83.064,169.385,37.597,157.070
C00724=1040.139,11.823,-83.048,169.383,37.596,157.070
C00725=1040.133,11.573,-83.033,169.381,37.595,157.069
C00726=1040.126,11.324,-83.018,169.379,37.595,157.069
C00727=1040.120,11.075,-83.003,169.377,37.594,157.069
C00728=1040.113,10.825,-82.988,169.376,37.594,157.069
C00729=1040.106,10.576,-82.972,169.374,37.594,157.069
C00730=1040.101,10.326,-82.957,169.372,37.593,157.069
C00731=1040.094,10.077,-82.941,169.369,37.593,157.069
C00732=1040.088,9.827,-82.926,169.367,37.592,157.069
C00733=1040.081,9.578,-82.911,169.365,37.591,157.068
C00734=1040.075,9.329,-82.896,169.363,37.591,157.068
C00735=1040.068,9.079,-82.881,169.361,37.590,157.068
C00736=1040.062,8.829,-82.866,169.359,37.590,157.068
C00737=1040.055,8.580,-82.850,169.357,37.589,157.068
C00738=1040.049,8.331,-82.835,169.355,37.589,157.068
C00739=1040.042,8.081,-82.820,169.353,37.588,157.068
C00740=1040.036,7.832,-82.804,169.351,37.587,157.068
C00741=1040.030,7.582,-82.789,169.348,37.587,157.067
C00742=1040.024,7.332,-82.774,169.346,37.586,157.067
C00743=1040.017,7.083,-82.759,169.344,37.586,157.067
C00744=1040.011,6.833,-82.743,169.342,37.585,157.067
C00745=1040.004,6.584,-82.728,169.340,37.584,157.067
C00746=1039.998,6.334,-82.713,169.338,37.584,157.067
C00747=1039.991,6.085,-82.698,169.336,37.583,157.067
C00748=1039.985,5.836,-82.683,169.334,37.583,157.066
C00749=1039.979,5.587,-82.668,169.332,37.582,157.066
C00750=1039.973,5.337,-82.653,169.330,37.581,157.066
C00751=1039.966,5.087,-82.638,169.328,37.581,157.066
C00752=1039.960,4.838,-82.622,169.325,37.580,157.066
C00753=1039.954,4.588,-82.607,169.323,37.580,157.066
C00754=1039.948,4.339,-82.592,169.321,37.579,157.066
C00755=1039.941,4.089,-82.577,169.319,37.579,157.066
C00756=1039.935,3.840,-82.563,169.317,37.577,157.065
C00757=1039.929,3.591,-82.547,169.315,37.577,157.065
C00758=1039.922,3.341,-82.532,169.313,37.576,157.065
C00759=1039.916,3.092,-82.517,169.311,37.576,157.065
C00760=1039.910,2.842,-82.502,169.309,37.575,157.065
C00761=1039.903,2.592,-82.487,169.306,37.574,157.065
C00762=1039.897,2.343,-82.472,169.304,37.574,157.064
C00763=1039.891,2.094,-82.458,169.302,37.573,157.064
C00764=1039.884,1.845,-82.442,169.300,37.573,157.064
C00765=1039.878,1.595,-82.427,169.298,37.572,157.064
C00766=1039.872,1.345,-82.412,169.296,37.571,157.064
C00767=1039.865,1.096,-82.397,169.294,37.571,157.064
C00768=1039.859,0.847,-82.383,169.292,37.570,157.064
C00769=1039.854,0.597,-82.367,169.290,37.570,157.064
C00770=1039.847,0.347,-82.352,169.288,37.569,157.063
C00771=1039.841,0.097,-82.337,169.285,37.569,157.063
C00772=1039.835,-0.152,-82.322,169.283,37.568,157.063
C00773=1039.829,-0.401,-82.308,169.281,37.567,157.063
C00774=1039.822,-0.651,-82.293,169.279,37.567,157.063
C00775=1039.816,-0.901,-82.278,169.277,37.566,157.063
C00776=1039.810,-1.150,-82.263,169.275,37.566,157.063
C00777=1039.804,-1.398,-82.248,169.273,37.565,157.063
C00778=1039.797,-1.648,-82.233,169.271,37.564,157.062
C00779=1039.791,-1.898,-82.218,169.269,37.564,157.062
C00780=1039.784,-2.147,-82.203,169.267,37.563,157.062
C00781=1039.779,-2.396,-82.188,169.265,37.563,157.062
C00782=1039.772,-2.646,-82.173,169.262,37.562,157.062
C00783=1039.766,-2.896,-82.159,169.260,37.561,157.062
C00784=1039.759,-3.179,-82.142,169.258,37.561,157.062
C00785=1039.752,-3.463,-82.125,169.256,37.560,157.061
C00786=1039.745,-3.746,-82.109,169.253,37.560,157.061
C00787=1039.737,-4.030,-82.091,169.251,37.559,157.061
C00788=1039.731,-4.279,-82.077,169.249,37.559,157.061
C00789=1039.725,-4.529,-82.063,169.247,37.558,157.061
C00790=1039.718,-4.779,-82.048,169.245,37.557,157.061
C00791=1039.712,-5.028,-82.033,169.243,37.557,157.061
C00792=1039.705,-5.277,-82.019,169.240,37.556,157.061
C00793=1039.699,-5.527,-82.004,169.238,37.556,157.061
C00794=1039.693,-5.776,-81.989,169.235,37.556,157.060
C00795=1039.686,-6.026,-81.976,169.233,37.555,157.060
C00796=1039.680,-6.275,-81.961,169.231,37.555,157.060
C00797=1039.674,-6.525,-81.946,169.229,37.554,157.060
C00798=1039.667,-6.774,-81.931,169.227,37.553,157.060
C00799=1039.660,-7.024,-81.917,169.225,37.553,157.060
C00800=1039.655,-7.273,-81.903,169.223,37.553,157.060
C00801=1039.648,-7.523,-81.888,169.221,37.552,157.060
C00802=1039.641,-7.772,-81.874,169.219,37.552,157.059
C00803=1039.635,-8.021,-81.859,169.217,37.551,157.059
C00804=1039.629,-8.272,-81.845,169.214,37.550,157.059
C00805=1039.622,-8.521,-81.830,169.212,37.551,157.059
C00806=1039.616,-8.770,-81.816,169.210,37.550,157.059
C00807=1039.610,-9.020,-81.801,169.208,37.549,157.059
C00808=1039.603,-9.270,-81.787,169.205,37.549,157.059
C00809=1039.598,-9.519,-81.773,169.203,37.548,157.059
C00810=1039.591,-9.768,-81.758,169.201,37.548,157.059
C00811=1039.584,-10.018,-81.744,169.199,37.548,157.059
C00812=1039.579,-10.267,-81.729,169.197,37.547,157.058
C00813=1039.572,-10.517,-81.715,169.195,37.546,157.058
C00814=1039.565,-10.767,-81.701,169.193,37.546,157.058
C00815=1039.560,-11.016,-81.686,169.191,37.545,157.058
C00816=1039.553,-11.265,-81.671,169.188,37.545,157.058
C00817=1039.546,-11.515,-81.658,169.186,37.544,157.058
C00818=1039.541,-11.764,-81.643,169.184,37.544,157.058
C00819=1039.534,-12.014,-81.628,169.182,37.544,157.058
C00820=1039.528,-12.263,-81.615,169.180,37.543,157.057
C00821=1039.522,-12.513,-81.600,169.177,37.542,157.057
C00822=1039.516,-12.763,-81.586,169.175,37.542,157.057
C00823=1039.509,-13.012,-81.572,169.173,37.541,157.057
C00824=1039.503,-13.261,-81.557,169.171,37.541,157.057
C00825=1039.497,-13.511,-81.543,169.169,37.541,157.057
C00826=1039.490,-13.760,-81.529,169.167,37.540,157.057
C00827=1039.484,-14.011,-81.514,169.165,37.540,157.057
C00828=1039.478,-14.260,-81.500,169.162,37.539,157.057
C00829=1039.471,-14.510,-81.486,169.160,37.538,157.056
C00830=1039.466,-14.758,-81.472,169.158,37.538,157.056
C00831=1039.459,-15.008,-81.457,169.156,37.538,157.056
C00832=1039.453,-15.257,-81.443,169.153,37.537,157.056
C00833=1039.447,-15.507,-81.428,169.151,37.537,157.056
C00834=1039.440,-15.757,-81.415,169.149,37.536,157.056
C00835=1039.434,-16.007,-81.401,169.147,37.536,157.056
C00836=1039.427,-16.256,-81.387,169.145,37.536,157.056
C00837=1039.421,-16.505,-81.373,169.143,37.535,157.056
C00838=1039.415,-16.755,-81.358,169.141,37.535,157.056
C00839=1039.408,-17.004,-81.345,169.138,37.534,157.055
C00840=1039.402,-17.254,-81.330,169.136,37.534,157.055
C00841=1039.395,-17.504,-81.316,169.134,37.534,157.055
C00842=1039.389,-17.753,-81.303,169.131,37.533,157.055
C00843=1039.383,-18.003,-81.288,169.129,37.533,157.055
C00844=1039.376,-18.252,-81.275,169.127,37.532,157.055
C00845=1039.370,-18.502,-81.260,169.125,37.532,157.055
C00846=1039.364,-18.751,-81.247,169.123,37.532,157.055
C00847=1039.357,-19.001,-81.233,169.120,37.531,157.055
C00848=1039.350,-19.282,-81.217,169.118,37.531,157.055
C00849=1039.342,-19.564,-81.201,169.116,37.530,157.054
C00850=1039.336,-19.847,-81.185,169.113,37.530,157.054
C00851=1039.329,-20.128,-81.170,169.111,37.529,157.054
C00852=1039.322,-20.378,-81.156,169.109,37.529,157.054
C00853=1039.316,-20.627,-81.143,169.106,37.529,157.054
C00854=1039.310,-20.877,-81.128,169.104,37.528,157.054
C00855=1039.303,-21.126,-81.114,169.101,37.528,157.054
C00856=1039.297,-21.376,-81.101,169.099,37.528,157.054
C00857=1039.291,-21.625,-81.087,169.097,37.527,157.054
C00858=1039.284,-21.875,-81.073,169.095,37.526,157.053
C00859=1039.279,-22.124,-81.059,169.092,37.527,157.053
C00860=1039.272,-22.374,-81.045,169.090,37.526,157.053
C00861=1039.265,-22.623,-81.031,169.088,37.525,157.053
C00862=1039.259,-22.873,-81.017,169.086,37.525,157.053
C00863=1039.253,-23.122,-81.004,169.084,37.525,157.053
C00864=1039.246,-23.372,-80.990,169.082,37.524,157.053
C00865=1039.241,-23.622,-80.976,169.080,37.524,157.053
C00866=1039.234,-23.871,-80.962,169.077,37.524,157.053
C00867=1039.227,-24.121,-80.949,169.075,37.523,157.053
C00868=1039.222,-24.370,-80.935,169.073,37.523,157.053
C00869=1039.215,-24.620,-80.921,169.071,37.523,157.053
C00870=1039.210,-24.870,-80.907,169.068,37.522,157.052
C00871=1039.203,-25.118,-80.893,169.066,37.521,157.052
C00872=1039.196,-25.368,-80.880,169.063,37.521,157.052
C00873=1039.191,-25.618,-80.866,169.061,37.521,157.052
C00874=1039.184,-25.868,-80.852,169.059,37.520,157.052
C00875=1039.178,-26.117,-80.839,169.057,37.520,157.052
C00876=1039.172,-26.367,-80.825,169.055,37.520,157.052
C00877=1039.165,-26.617,-80.811,169.053,37.519,157.052
C00878=1039.159,-26.866,-80.798,169.050,37.519,157.052
C00879=1039.154,-27.115,-80.784,169.048,37.519,157.052
C00880=1039.147,-27.365,-80.770,169.046,37.518,157.051
C00881=1039.140,-27.614,-80.757,169.044,37.518,157.051
C00882=1039.134,-27.864,-80.743,169.042,37.518,157.051
C00883=1039.127,-28.113,-80.730,169.039,37.518,157.051
C00884=1039.121,-28.363,-80.716,169.037,37.517,157.051
C00885=1039.114,-28.613,-80.703,169.035,37.517,157.051
C00886=1039.108,-28.862,-80.689,169.032,37.516,157.051
C00887=1039.101,-29.112,-80.676,169.029,37.517,157.051
C00888=1039.095,-29.361,-80.663,169.027,37.516,157.051
C00889=1039.090,-29.611,-80.649,169.025,37.516,157.051
C00890=1039.083,-29.861,-80.636,169.023,37.515,157.051
C00891=1039.077,-30.110,-80.622,169.021,37.515,157.051
C00892=1039.071,-30.360,-80.609,169.018,37.515,157.051
C00893=1039.064,-30.610,-80.596,169.016,37.514,157.050
C00894=1039.058,-30.859,-80.582,169.014,37.514,157.050
C00895=1039.051,-31.108,-80.569,169.012,37.514,157.050
C00896=1039.045,-31.358,-80.555,169.009,37.514,157.050
C00897=1039.038,-31.607,-80.542,169.007,37.513,157.050
C00898=1039.032,-31.857,-80.529,169.005,37.513,157.050
C00899=1039.025,-32.107,-80.515,169.003,37.513,157.050
C00900=1039.019,-32.356,-80.502,169.001,37.513,157.050
C00901=1039.013,-32.605,-80.489,168.998,37.512,157.050
C00902=1039.008,-32.855,-80.476,168.996,37.512,157.050
C00903=1039.001,-33.105,-80.462,168.994,37.512,157.050
C00904=1038.995,-33.355,-80.449,168.992,37.512,157.050
C00905=1038.989,-33.604,-80.435,168.988,37.511,157.050
C00906=1038.982,-33.853,-80.422,168.986,37.511,157.050
C00907=1038.975,-34.103,-80.408,168.984,37.511,157.049
C00908=1038.970,-34.353,-80.396,168.982,37.511,157.049
C00909=1038.963,-34.602,-80.383,168.979,37.510,157.049
C00910=1038.957,-34.851,-80.369,168.977,37.510,157.049
C00911=1038.950,-35.101,-80.356,168.975,37.510,157.049
C00912=1038.944,-35.382,-80.342,168.972,37.509,157.049
C00913=1038.937,-35.663,-80.326,168.970,37.509,157.049
C00914=1038.929,-35.945,-80.311,168.967,37.508,157.049
C00915=1038.922,-36.226,-80.296,168.965,37.508,157.049
C00916=1038.916,-36.476,-80.283,168.963,37.508,157.049
C00917=1038.910,-36.725,-80.270,168.960,37.508,157.049
C00918=1038.904,-36.974,-80.257,168.958,37.507,157.049
C00919=1038.898,-37.223,-80.243,168.956,37.507,157.049
C00920=1038.891,-37.474,-80.230,168.954,37.507,157.048
C00921=1038.885,-37.723,-80.217,168.951,37.507,157.048
C00922=1038.879,-37.973,-80.204,168.949,37.506,157.048
C00923=1038.873,-38.222,-80.191,168.947,37.506,157.048
C00924=1038.867,-38.472,-80.178,168.944,37.506,157.048
C00925=1038.860,-38.722,-80.164,168.941,37.506,157.048
C00926=1038.854,-38.972,-80.152,168.939,37.505,157.048
C00927=1038.848,-39.221,-80.139,168.937,37.505,157.048
C00928=1038.841,-39.470,-80.126,168.934,37.505,157.048
C00929=1038.835,-39.720,-80.113,168.932,37.505,157.048
C00930=1038.828,-39.970,-80.100,168.930,37.505,157.048
C00931=1038.822,-40.220,-80.087,168.928,37.504,157.048
C00932=1038.816,-40.469,-80.074,168.925,37.504,157.048
C00933=1038.809,-40.718,-80.061,168.923,37.504,157.048
C00934=1038.803,-40.968,-80.049,168.921,37.504,157.047
C00935=1038.797,-41.217,-80.035,168.918,37.504,157.047
C00936=1038.790,-41.467,-80.023,168.916,37.504,157.047
C00937=1038.784,-41.717,-80.009,168.914,37.503,157.047
C00938=1038.778,-41.966,-79.997,168.911,37.503,157.047
C00939=1038.771,-42.216,-79.984,168.909,37.503,157.047
C00940=1038.765,-42.465,-79.971,168.907,37.503,157.047
C00941=1038.759,-42.715,-79.958,168.905,37.503,157.047
C00942=1038.753,-42.964,-79.946,168.902,37.502,157.047
C00943=1038.746,-43.214,-79.933,168.900,37.502,157.047
C00944=1038.740,-43.464,-79.920,168.898,37.502,157.047
C00945=1038.734,-43.713,-79.907,168.895,37.502,157.047
C00946=1038.727,-43.963,-79.895,168.893,37.502,157.047
C00947=1038.721,-44.212,-79.882,168.891,37.502,157.047
C00948=1038.715,-44.462,-79.869,168.887,37.501,157.047
C00949=1038.709,-44.712,-79.856,168.885,37.501,157.047
C00950=1038.703,-44.961,-79.843,168.883,37.501,157.047
C00951=1038.696,-45.211,-79.831,168.880,37.501,157.047
C00952=1038.690,-45.460,-79.818,168.878,37.501,157.046
C00953=1038.684,-45.710,-79.805,168.876,37.501,157.046
C00954=1038.678,-45.959,-79.792,168.874,37.500,157.046
C00955=1038.671,-46.209,-79.780,168.871,37.500,157.046
C00956=1038.665,-46.459,-79.768,168.869,37.501,157.046
C00957=1038.659,-46.708,-79.754,168.867,37.500,157.046
C00958=1038.652,-46.958,-79.742,168.864,37.500,157.046
C00959=1038.646,-47.208,-79.729,168.862,37.500,157.046
C00960=1038.640,-47.457,-79.716,168.860,37.499,157.046
C00961=1038.634,-47.707,-79.704,168.857,37.500,157.046
C00962=1038.627,-47.957,-79.692,168.855,37.500,157.046
C00963=1038.621,-48.206,-79.678,168.853,37.499,157.046
C00964=1038.615,-48.456,-79.666,168.850,37.499,157.046
C00965=1038.609,-48.706,-79.653,168.848,37.499,157.046
C00966=1038.602,-48.955,-79.641,168.846,37.499,157.046
C00967=1038.596,-49.205,-79.628,168.843,37.499,157.046
C00968=1038.591,-49.454,-79.616,168.841,37.499,157.046
C00969=1038.585,-49.704,-79.603,168.839,37.499,157.046
C00970=1038.578,-49.953,-79.591,168.836,37.498,157.046
C00971=1038.572,-50.203,-79.578,168.834,37.498,157.046
C00972=1038.566,-50.453,-79.566,168.832,37.498,157.045
C00973=1038.560,-50.702,-79.554,168.829,37.498,157.045
C00974=1038.553,-50.951,-79.540,168.827,37.498,157.045
C00975=1038.547,-51.201,-79.528,168.824,37.498,157.045
C00976=1038.540,-51.483,-79.515,168.821,37.498,157.045
C00977=1038.532,-51.764,-79.501,168.818,37.498,157.045
C00978=1038.525,-52.046,-79.487,168.815,37.498,157.045
C00979=1038.517,-52.328,-79.473,168.813,37.498,157.045
C00980=1038.511,-52.577,-79.461,168.810,37.498,157.045
C00981=1038.505,-52.827,-79.448,168.808,37.498,157.045
C00982=1038.498,-53.077,-79.436,168.805,37.498,157.045
C00983=1038.492,-53.326,-79.424,168.803,37.498,157.045
C00984=1038.486,-53.575,-79.412,168.801,37.498,157.045
C00985=1038.479,-53.825,-79.400,168.798,37.498,157.045
C00986=1038.473,-54.075,-79.388,168.796,37.498,157.045
C00987=1038.467,-54.324,-79.376,168.793,37.498,157.045
C00988=1038.460,-54.574,-79.364,168.791,37.498,157.045
C00989=1038.454,-54.824,-79.351,168.789,37.498,157.045
C00990=1038.448,-55.073,-79.339,168.786,37.498,157.045
C00991=1038.441,-55.323,-79.327,168.784,37.498,157.045
C00992=1038.435,-55.573,-79.315,168.781,37.498,157.045
C00993=1038.428,-55.822,-79.303,168.779,37.498,157.045
C00994=1038.422,-56.072,-79.291,168.777,37.498,157.045
C00995=1038.416,-56.322,-79.278,168.774,37.498,157.045
C00996=1038.409,-56.571,-79.266,168.772,37.498,157.045
C00997=1038.403,-56.821,-79.254,168.769,37.499,157.045
C00998=1038.397,-57.070,-79.242,168.767,37.499,157.045
C00999=1038.391,-57.320,-79.230,168.765,37.499,157.045
C01000=1038.384,-57.569,-79.218,168.762,37.499,157.045
C01001=1038.378,-57.819,-79.206,168.760,37.499,157.045
C01002=1038.371,-58.069,-79.194,168.757,37.499,157.045
C01003=1038.365,-58.318,-79.182,168.755,37.498,157.045
C01004=1038.359,-58.568,-79.169,168.752,37.498,157.045
C01005=1038.353,-58.817,-79.157,168.750,37.498,157.045
C01006=1038.346,-59.067,-79.146,168.748,37.498,157.045
C01007=1038.341,-59.317,-79.134,168.745,37.499,157.045
C01008=1038.334,-59.567,-79.122,168.743,37.499,157.045
C01009=1038.327,-59.816,-79.110,168.740,37.499,157.045
C01010=1038.321,-60.066,-79.097,168.738,37.499,157.045
C01011=1038.315,-60.315,-79.086,168.735,37.499,157.045
C01012=1038.309,-60.565,-79.074,168.733,37.499,157.045
C01013=1038.303,-60.815,-79.061,168.731,37.499,157.044
C01014=1038.296,-61.065,-79.050,168.728,37.499,157.044
C01015=1038.290,-61.314,-79.038,168.726,37.499,157.044
C01016=1038.284,-61.563,-79.026,168.723,37.499,157.044
C01017=1038.278,-61.813,-79.014,168.721,37.499,157.044
C01018=1038.271,-62.063,-79.002,168.718,37.499,157.044
C01019=1038.265,-62.313,-78.991,168.716,37.499,157.044
C01020=1038.259,-62.563,-78.978,168.714,37.499,157.044
C01021=1038.253,-62.812,-78.966,168.711,37.499,157.044
C01022=1038.246,-63.061,-78.954,168.709,37.499,157.044
C01023=1038.241,-63.312,-78.943,168.706,37.500,157.044
C01024=1038.234,-63.561,-78.931,168.704,37.500,157.044
C01025=1038.228,-63.810,-78.919,168.701,37.500,157.044
C01026=1038.221,-64.060,-78.907,168.699,37.500,157.044
C01027=1038.216,-64.310,-78.895,168.697,37.500,157.044
C01028=1038.210,-64.559,-78.884,168.694,37.500,157.044
C01029=1038.203,-64.809,-78.872,168.692,37.500,157.044
C01030=1038.197,-65.059,-78.860,168.689,37.500,157.044
C01031=1038.191,-65.309,-78.848,168.687,37.500,157.044
C01032=1038.185,-65.558,-78.836,168.684,37.500,157.044
C01033=1038.178,-65.808,-78.825,168.682,37.500,157.044
C01034=1038.172,-66.058,-78.813,168.679,37.500,157.044
C01035=1038.166,-66.306,-78.801,168.677,37.500,157.044
C01036=1038.160,-66.557,-78.790,168.675,37.500,157.044
C01037=1038.153,-66.806,-78.778,168.672,37.500,157.044
C01038=1038.148,-67.055,-78.766,168.670,37.500,157.044
C01039=1038.142,-67.306,-78.754,168.667,37.501,157.044
C01040=1038.135,-67.588,-78.741,168.664,37.501,157.044
C01041=1038.127,-67.871,-78.727,168.662,37.501,157.044
C01042=1038.121,-68.154,-78.714,168.659,37.501,157.044
C01043=1038.114,-68.436,-78.701,168.656,37.501,157.044
C01044=1038.108,-68.687,-78.690,168.654,37.501,157.044
C01045=1038.101,-68.935,-78.678,168.651,37.501,157.044
C01046=1038.096,-69.185,-78.666,168.649,37.501,157.044
C01047=1038.089,-69.436,-78.655,168.646,37.501,157.044
C01048=1038.083,-69.684,-78.643,168.644,37.501,157.044
C01049=1038.077,-69.935,-78.632,168.641,37.501,157.044
C01050=1038.072,-70.184,-78.620,168.639,37.501,157.044
C01051=1038.065,-70.434,-78.608,168.636,37.501,157.044
C01052=1038.059,-70.684,-78.596,168.634,37.501,157.044
C01053=1038.053,-70.933,-78.585,168.631,37.502,157.044
C01054=1038.047,-71.183,-78.573,168.629,37.502,157.044
C01055=1038.041,-71.432,-78.562,168.627,37.502,157.044
C01056=1038.035,-71.682,-78.550,168.624,37.502,157.044
C01057=1038.029,-71.931,-78.539,168.622,37.502,157.044
C01058=1038.022,-72.181,-78.527,168.619,37.502,157.044
C01059=1038.017,-72.431,-78.516,168.617,37.503,157.044
C01060=1038.011,-72.681,-78.505,168.614,37.503,157.044
C01061=1038.005,-72.930,-78.493,168.612,37.503,157.044
C01062=1037.998,-73.180,-78.482,168.609,37.503,157.044
C01063=1037.992,-73.430,-78.470,168.607,37.503,157.044
C01064=1037.987,-73.679,-78.458,168.604,37.503,157.044
C01065=1037.980,-73.930,-78.447,168.602,37.503,157.044
C01066=1037.974,-74.179,-78.435,168.599,37.503,157.044
C01067=1037.968,-74.429,-78.424,168.597,37.503,157.044
C01068=1037.962,-74.678,-78.413,168.594,37.504,157.044
C01069=1037.956,-74.928,-78.401,168.592,37.504,157.044
C01070=1037.950,-75.177,-78.390,168.589,37.504,157.044
C01071=1037.944,-75.427,-78.379,168.587,37.504,157.044
C01072=1037.938,-75.676,-78.368,168.584,37.505,157.044
C01073=1037.931,-75.927,-78.356,168.582,37.505,157.044
C01074=1037.925,-76.176,-78.346,168.579,37.505,157.044
C01075=1037.918,-76.426,-78.335,168.577,37.505,157.044
C01076=1037.912,-76.675,-78.323,168.574,37.506,157.044
C01077=1037.906,-76.925,-78.312,168.572,37.506,157.044
C01078=1037.900,-77.174,-78.301,168.569,37.506,157.044
C01079=1037.894,-77.425,-78.290,168.567,37.506,157.044
C01080=1037.888,-77.674,-78.278,168.564,37.507,157.044
C01081=1037.882,-77.924,-78.267,168.562,37.507,157.044
C01082=1037.876,-78.173,-78.256,168.559,37.507,157.044
C01083=1037.869,-78.423,-78.245,168.556,37.507,157.044
C01084=1037.864,-78.673,-78.234,168.554,37.507,157.044
C01085=1037.857,-78.923,-78.223,168.551,37.508,157.044
C01086=1037.851,-79.172,-78.211,168.549,37.508,157.044
C01087=1037.844,-79.422,-78.201,168.546,37.508,157.044
C01088=1037.838,-79.671,-78.190,168.544,37.508,157.044
C01089=1037.833,-79.921,-78.179,168.541,37.508,157.044
C01090=1037.826,-80.171,-78.168,168.539,37.509,157.044
C01091=1037.821,-80.420,-78.157,168.536,37.509,157.044
C01092=1037.814,-80.670,-78.146,168.534,37.510,157.044
C01093=1037.808,-80.920,-78.135,168.531,37.510,157.044
C01094=1037.802,-81.170,-78.124,168.528,37.510,157.044
C01095=1037.795,-81.419,-78.114,168.526,37.511,157.044
C01096=1037.789,-81.669,-78.102,168.523,37.511,157.044
C01097=1037.783,-81.919,-78.092,168.521,37.512,157.044
C01098=1037.776,-82.169,-78.081,168.518,37.512,157.044
C01099=1037.770,-82.418,-78.070,168.516,37.512,157.044
C01100=1037.764,-82.668,-78.059,168.513,37.512,157.044
C01101=1037.757,-82.918,-78.048,168.510,37.513,157.045
C01102=1037.752,-83.167,-78.038,168.508,37.513,157.045
C01103=1037.745,-83.417,-78.026,168.505,37.514,157.045
C01104=1037.738,-83.701,-78.014,168.502,37.514,157.045
C01105=1037.731,-83.987,-78.001,168.499,37.515,157.045
C01106=1037.724,-84.271,-77.989,168.496,37.515,157.045
C01107=1037.717,-84.557,-77.977,168.494,37.516,157.045
C01108=1037.711,-84.806,-77.966,168.492,37.516,157.045
C01109=1037.704,-85.056,-77.956,168.489,37.516,157.045
C01110=1037.698,-85.306,-77.945,168.487,37.516,157.045
C01111=1037.692,-85.555,-77.935,168.484,37.517,157.045
C01112=1037.685,-85.805,-77.923,168.481,37.517,157.045
C01113=1037.680,-86.054,-77.912,168.479,37.518,157.045
C01114=1037.674,-86.304,-77.903,168.476,37.518,157.045
C01115=1037.667,-86.554,-77.892,168.474,37.519,157.045
C01116=1037.661,-86.804,-77.881,168.471,37.519,157.045
C01117=1037.655,-87.053,-77.870,168.469,37.520,157.045
C01118=1037.649,-87.303,-77.859,168.466,37.520,157.045
C01119=1037.643,-87.553,-77.848,168.463,37.520,157.045
C01120=1037.637,-87.803,-77.839,168.461,37.520,157.045
C01121=1037.630,-88.053,-77.827,168.458,37.521,157.045
C01122=1037.624,-88.302,-77.817,168.456,37.521,157.045
C01123=1037.618,-88.551,-77.806,168.453,37.522,157.045
C01124=1037.612,-88.801,-77.795,168.450,37.523,157.045
C01125=1037.606,-89.051,-77.786,168.448,37.523,157.045
C01126=1037.600,-89.301,-77.775,168.445,37.523,157.046
C01127=1037.593,-89.550,-77.764,168.443,37.524,157.046
C01128=1037.587,-89.800,-77.753,168.440,37.524,157.046
C01129=1037.581,-90.050,-77.742,168.437,37.524,157.046
C01130=1037.575,-90.300,-77.733,168.435,37.525,157.046
C01131=1037.569,-90.549,-77.722,168.432,37.525,157.046
C01132=1037.563,-90.798,-77.712,168.430,37.526,157.046
C01133=1037.557,-91.049,-77.701,168.427,37.526,157.046
C01134=1037.551,-91.299,-77.690,168.424,37.527,157.046
C01135=1037.545,-91.548,-77.680,168.422,37.527,157.046
C01136=1037.539,-91.797,-77.669,168.420,37.527,157.046
C01137=1037.532,-92.048,-77.659,168.418,37.528,157.046
C01138=1037.526,-92.297,-77.648,168.415,37.528,157.046
C01139=1037.521,-92.547,-77.637,168.412,37.529,157.046
C01140=1037.515,-92.796,-77.628,168.410,37.529,157.046
C01141=1037.509,-93.046,-77.617,168.407,37.530,157.046
C01142=1037.503,-93.296,-77.607,168.404,37.530,157.046
C01143=1037.496,-93.546,-77.596,168.402,37.531,157.046
C01144=1037.490,-93.795,-77.586,168.399,37.531,157.046
C01145=1037.484,-94.045,-77.576,168.397,37.531,157.046
C01146=1037.479,-94.295,-77.565,168.394,37.532,157.046
C01147=1037.472,-94.544,-77.554,168.391,37.532,157.046
C01148=1037.467,-94.794,-77.544,168.389,37.533,157.047
C01149=1037.460,-95.044,-77.534,168.386,37.533,157.047
C01150=1037.454,-95.294,-77.523,168.384,37.534,157.047
C01151=1037.448,-95.543,-77.513,168.381,37.534,157.047
C01152=1037.442,-95.793,-77.503,168.378,37.535,157.047
C01153=1037.436,-96.042,-77.493,168.376,37.535,157.047
C01154=1037.430,-96.292,-77.482,168.373,37.535,157.047
C01155=1037.425,-96.542,-77.472,168.371,37.536,157.047
C01156=1037.418,-96.791,-77.461,168.368,37.537,157.047
C01157=1037.413,-97.041,-77.451,168.365,37.537,157.047
C01158=1037.406,-97.292,-77.441,168.363,37.538,157.047
C01159=1037.400,-97.541,-77.430,168.361,37.538,157.047
C01160=1037.394,-97.791,-77.421,168.357,37.538,157.047
C01161=1037.388,-98.040,-77.411,168.356,37.539,157.047
C01162=1037.382,-98.290,-77.400,168.353,37.540,157.047
C01163=1037.376,-98.540,-77.390,168.350,37.541,157.047
C01164=1037.370,-98.789,-77.381,168.348,37.541,157.047
C01165=1037.364,-99.040,-77.370,168.345,37.541,157.048
C01166=1037.358,-99.289,-77.360,168.342,37.542,157.048
C01167=1037.351,-99.539,-77.350,168.340,37.543,157.048
///RCONF 1,0,0,0,1,0,0,0,0,0,0,0,0,0,0,0,0,0,0,0,0,0,0,0
C01168=1037.345,-99.826,-77.339,168.337,37.544,157.048
C01169=1037.337,-100.113,-77.327,168.334,37.544,157.048
C01170=1037.330,-100.400,-77.316,168.331,37.545,157.048
C01171=1037.323,-100.688,-77.304,168.327,37.546,157.048
C01172=1037.317,-100.938,-77.294,168.325,37.546,157.048
C01173=1037.311,-101.187,-77.284,168.322,37.547,157.048
C01174=1037.305,-101.437,-77.274,168.319,37.547,157.048
C01175=1037.299,-101.687,-77.264,168.317,37.548,157.048
C01176=1037.293,-101.936,-77.254,168.315,37.549,157.048
C01177=1037.286,-102.186,-77.244,168.312,37.550,157.049
C01178=1037.281,-102.436,-77.234,168.310,37.550,157.049
C01179=1037.275,-102.686,-77.225,168.307,37.550,157.049
C01180=1037.268,-102.935,-77.214,168.304,37.551,157.049
C01181=1037.262,-103.185,-77.205,168.302,37.552,157.049
C01182=1037.257,-103.435,-77.195,168.299,37.553,157.049
C01183=1037.251,-103.684,-77.185,168.296,37.553,157.049
C01184=1037.244,-103.934,-77.175,168.294,37.553,157.049
C01185=1037.238,-104.183,-77.165,168.291,37.554,157.049
C01186=1037.233,-104.434,-77.155,168.288,37.555,157.049
C01187=1037.226,-104.683,-77.145,168.286,37.556,157.049
C01188=1037.220,-104.933,-77.136,168.283,37.556,157.049
C01189=1037.214,-105.182,-77.126,168.280,37.557,157.049
C01190=1037.208,-105.432,-77.115,168.278,37.558,157.050
C01191=1037.202,-105.682,-77.106,168.276,37.558,157.050
C01192=1037.196,-105.932,-77.096,168.273,37.559,157.050
C01193=1037.190,-106.182,-77.087,168.271,37.559,157.050
C01194=1037.184,-106.432,-77.077,168.268,37.560,157.050
C01195=1037.178,-106.682,-77.067,168.265,37.561,157.050
C01196=1037.172,-106.931,-77.057,168.263,37.561,157.050
C01197=1037.166,-107.181,-77.047,168.260,37.562,157.050
C01198=1037.159,-107.430,-77.038,168.257,37.563,157.050
C01199=1037.154,-107.680,-77.028,168.255,37.564,157.050
C01200=1037.148,-107.929,-77.019,168.252,37.564,157.050
C01201=1037.141,-108.179,-77.009,168.249,37.565,157.050
C01202=1037.136,-108.429,-76.999,168.246,37.566,157.051
C01203=1037.130,-108.679,-76.989,168.244,37.567,157.051
C01204=1037.124,-108.929,-76.980,168.241,37.567,157.051
C01205=1037.117,-109.179,-76.970,168.238,37.568,157.051
C01206=1037.111,-109.428,-76.961,168.237,37.569,157.051
C01207=1037.105,-109.678,-76.951,168.234,37.570,157.051
C01208=1037.099,-109.928,-76.942,168.231,37.570,157.051
C01209=1037.093,-110.177,-76.932,168.228,37.571,157.051
C01210=1037.087,-110.427,-76.923,168.226,37.572,157.051
C01211=1037.081,-110.677,-76.913,168.223,37.573,157.051
C01212=1037.075,-110.927,-76.904,168.220,37.573,157.051
C01213=1037.069,-111.176,-76.894,168.218,37.574,157.052
C01214=1037.063,-111.426,-76.885,168.215,37.575,157.052
C01215=1037.056,-111.676,-76.875,168.212,37.576,157.052
C01216=1037.051,-111.925,-76.866,168.209,37.577,157.052
C01217=1037.045,-112.175,-76.856,168.207,37.578,157.052
C01218=1037.038,-112.425,-76.847,168.205,37.578,157.052
C01219=1037.033,-112.675,-76.838,168.202,37.579,157.052
C01220=1037.026,-112.925,-76.828,168.200,37.580,157.052
C01221=1037.020,-113.175,-76.819,168.197,37.581,157.052
C01222=1037.015,-113.424,-76.809,168.194,37.581,157.053
C01223=1037.008,-113.674,-76.800,168.191,37.582,157.053
C01224=1037.002,-113.923,-76.790,168.189,37.583,157.053
C01225=1036.997,-114.173,-76.780,168.186,37.583,157.053
C01226=1036.990,-114.424,-76.772,168.183,37.584,157.053
C01227=1036.985,-114.673,-76.763,168.181,37.586,157.053
C01228=1036.979,-114.922,-76.753,168.178,37.586,157.053
C01229=1036.972,-115.172,-76.744,168.175,37.587,157.053
C01230=1036.966,-115.422,-76.734,168.173,37.588,157.053
C01231=1036.960,-115.672,-76.725,168.171,37.589,157.054
C01232=1036.954,-115.958,-76.715,168.167,37.590,157.054
C01233=1036.947,-116.245,-76.704,168.164,37.591,157.054
C01234=1036.940,-116.531,-76.694,168.161,37.592,157.054
C01235=1036.933,-116.818,-76.683,168.158,37.593,157.054
C01236=1036.927,-117.068,-76.673,168.155,37.594,157.054
C01237=1036.920,-117.317,-76.664,168.153,37.594,157.054
C01238=1036.915,-117.567,-76.656,168.150,37.595,157.054
C01239=1036.909,-117.817,-76.646,168.147,37.596,157.054
C01240=1036.903,-118.066,-76.636,168.145,37.597,157.055
C01241=1036.897,-118.316,-76.627,168.143,37.598,157.055
C01242=1036.891,-118.566,-76.618,168.140,37.599,157.055
C01243=1036.885,-118.816,-76.609,168.137,37.600,157.055
C01244=1036.878,-119.065,-76.600,168.134,37.601,157.055
C01245=1036.873,-119.315,-76.591,168.132,37.602,157.055
C01246=1036.867,-119.565,-76.582,168.129,37.602,157.055
C01247=1036.861,-119.815,-76.573,168.126,37.603,157.055
C01248=1036.855,-120.064,-76.564,168.123,37.605,157.056
C01249=1036.849,-120.314,-76.554,168.121,37.605,157.056
C01250=1036.843,-120.564,-76.546,168.119,37.606,157.056
C01251=1036.837,-120.813,-76.537,168.116,37.607,157.056
C01252=1036.831,-121.064,-76.528,168.113,37.608,157.056
C01253=1036.825,-121.314,-76.518,168.111,37.609,157.056
C01254=1036.819,-121.563,-76.509,168.108,37.610,157.056
C01255=1036.813,-121.813,-76.501,168.105,37.611,157.057
C01256=1036.807,-122.063,-76.491,168.102,37.612,157.057
C01257=1036.801,-122.312,-76.483,168.100,37.613,157.057
C01258=1036.795,-122.562,-76.473,168.097,37.613,157.057
C01259=1036.789,-122.812,-76.464,168.094,37.615,157.057
C01260=1036.783,-123.061,-76.456,168.092,37.615,157.057
C01261=1036.777,-123.312,-76.447,168.089,37.616,157.057
C01262=1036.772,-123.561,-76.438,168.087,37.618,157.057
C01263=1036.766,-123.811,-76.429,168.084,37.618,157.057
C01264=1036.759,-124.061,-76.420,168.081,37.619,157.058
C01265=1036.753,-124.310,-76.411,168.078,37.621,157.058
C01266=1036.747,-124.560,-76.402,168.076,37.621,157.058
C01267=1036.742,-124.810,-76.393,168.073,37.623,157.058
C01268=1036.735,-125.060,-76.385,168.070,37.623,157.058
C01269=1036.729,-125.310,-76.376,168.067,37.624,157.058
C01270=1036.724,-125.559,-76.367,168.066,37.626,157.058
C01271=1036.717,-125.809,-76.358,168.063,37.626,157.059
C01272=1036.712,-126.059,-76.350,168.060,37.628,157.059
C01273=1036.705,-126.309,-76.341,168.057,37.628,157.059
C01274=1036.699,-126.559,-76.332,168.054,37.630,157.059
C01275=1036.694,-126.808,-76.323,168.052,37.631,157.059
C01276=1036.687,-127.058,-76.314,168.049,37.631,157.059
C01277=1036.682,-127.308,-76.306,168.046,37.633,157.059
C01278=1036.676,-127.558,-76.297,168.044,37.634,157.060
C01279=1036.669,-127.807,-76.288,168.041,37.635,157.060
C01280=1036.664,-128.056,-76.280,168.039,37.636,157.060
C01281=1036.660,-128.306,-76.270,168.036,37.636,157.060
C01282=1036.656,-128.556,-76.259,168.034,37.636,157.060
C01283=1036.653,-128.806,-76.248,168.032,37.635,157.060
C01284=1036.650,-129.056,-76.237,168.029,37.634,157.059
C01285=1036.649,-129.306,-76.225,168.027,37.632,157.059
C01286=1036.647,-129.556,-76.212,168.025,37.630,157.059
C01287=1036.647,-129.805,-76.199,168.024,37.627,157.058
C01288=1036.648,-130.056,-76.184,168.021,37.625,157.058
C01289=1036.649,-130.305,-76.170,168.020,37.621,157.057
C01290=1036.651,-130.555,-76.156,168.018,37.618,157.057
C01291=1036.653,-130.805,-76.140,168.017,37.613,157.056
C01292=1036.657,-131.056,-76.124,168.016,37.608,157.055
C01293=1036.661,-131.306,-76.107,168.014,37.603,157.054
C01294=1036.666,-131.556,-76.089,168.014,37.598,157.053
C01295=1036.673,-131.806,-76.071,168.012,37.591,157.052
C01296=1036.335,-131.830,-76.345,167.964,37.802,157.087
C01297=1036.329,-131.581,-76.363,167.965,37.808,157.088
C01298=1036.324,-131.330,-76.381,167.966,37.814,157.089
C01299=1036.319,-131.081,-76.398,167.968,37.819,157.090
C01300=1036.317,-130.830,-76.414,167.969,37.824,157.091
C01301=1036.314,-130.580,-76.430,167.970,37.828,157.091
C01302=1036.311,-130.330,-76.445,167.971,37.832,157.092
C01303=1036.310,-130.080,-76.459,167.974,37.836,157.093
C01304=1036.310,-129.830,-76.473,167.975,37.839,157.093
C01305=1036.310,-129.580,-76.487,167.977,37.841,157.093
C01306=1036.311,-129.331,-76.499,167.979,37.843,157.094
C01307=1036.313,-129.081,-76.511,167.981,37.845,157.094
C01308=1036.315,-128.830,-76.523,167.983,37.846,157.094
C01309=1036.319,-128.580,-76.534,167.985,37.847,157.095
C01310=1036.322,-128.330,-76.545,167.987,37.847,157.095
C01311=1036.327,-128.081,-76.554,167.991,37.846,157.095
C01312=1036.332,-127.831,-76.563,167.993,37.846,157.095
C01313=1036.338,-127.582,-76.572,167.995,37.845,157.094
C01314=1036.344,-127.332,-76.580,167.998,37.843,157.094
C01315=1036.349,-127.082,-76.589,168.001,37.843,157.094
C01316=1036.356,-126.833,-76.598,168.004,37.841,157.094
C01317=1036.362,-126.583,-76.606,168.007,37.841,157.094
C01318=1036.368,-126.333,-76.616,168.009,37.839,157.094
C01319=1036.373,-126.084,-76.624,168.012,37.838,157.094
C01320=1036.380,-125.834,-76.633,168.014,37.837,157.093
C01321=1036.386,-125.584,-76.642,168.017,37.836,157.093
C01322=1036.392,-125.334,-76.650,168.020,37.835,157.093
C01323=1036.398,-125.084,-76.659,168.022,37.834,157.093
C01324=1036.403,-124.835,-76.668,168.025,37.833,157.093
C01325=1036.410,-124.585,-76.676,168.028,37.832,157.093
C01326=1036.415,-124.336,-76.686,168.031,37.831,157.093
C01327=1036.421,-124.085,-76.694,168.034,37.830,157.092
C01328=1036.427,-123.835,-76.704,168.036,37.829,157.092
C01329=1036.433,-123.586,-76.712,168.038,37.827,157.092
C01330=1036.440,-123.336,-76.722,168.041,37.827,157.092
C01331=1036.445,-123.087,-76.730,168.044,37.826,157.092
C01332=1036.451,-122.837,-76.740,168.046,37.824,157.092
C01333=1036.457,-122.586,-76.748,168.049,37.824,157.092
C01334=1036.463,-122.338,-76.757,168.052,37.823,157.092
C01335=1036.469,-122.087,-76.766,168.055,37.822,157.091
C01336=1036.475,-121.837,-76.775,168.058,37.821,157.091
C01337=1036.481,-121.588,-76.784,168.060,37.820,157.091
C01338=1036.487,-121.338,-76.793,168.062,37.819,157.091
C01339=1036.493,-121.088,-76.802,168.065,37.818,157.091
C01340=1036.499,-120.839,-76.811,168.068,37.817,157.091
C01341=1036.505,-120.588,-76.820,168.070,37.816,157.091
C01342=1036.511,-120.338,-76.829,168.073,37.815,157.091
C01343=1036.516,-120.089,-76.839,168.076,37.814,157.090
C01344=1036.523,-119.839,-76.847,168.079,37.813,157.090
C01345=1036.529,-119.589,-76.856,168.082,37.812,157.090
C01346=1036.535,-119.340,-76.866,168.084,37.811,157.090
C01347=1036.541,-119.090,-76.874,168.087,37.810,157.090
C01348=1036.547,-118.840,-76.884,168.089,37.809,157.090
C01349=1036.552,-118.590,-76.893,168.092,37.808,157.090
C01350=1036.559,-118.341,-76.901,168.094,37.808,157.090
C01351=1036.565,-118.091,-76.911,168.097,37.806,157.089
C01352=1036.570,-117.841,-76.920,168.100,37.805,157.089
C01353=1036.577,-117.592,-76.929,168.103,37.805,157.089
C01354=1036.583,-117.342,-76.939,168.105,37.804,157.089
C01355=1036.589,-117.092,-76.948,168.108,37.802,157.089
C01356=1036.594,-116.842,-76.957,168.111,37.802,157.089
C01357=1036.602,-116.556,-76.967,168.113,37.801,157.089
C01358=1036.608,-116.269,-76.978,168.116,37.799,157.089
C01359=1036.615,-115.983,-76.989,168.119,37.799,157.088
C01360=1036.623,-115.696,-76.999,168.123,37.798,157.088
C01361=1036.629,-115.447,-77.009,168.125,37.796,157.088
C01362=1036.635,-115.197,-77.018,168.128,37.796,157.088
C01363=1036.640,-114.947,-77.027,168.131,37.795,157.088
C01364=1036.646,-114.697,-77.036,168.134,37.794,157.088
C01365=1036.653,-114.448,-77.046,168.136,37.793,157.088
C01366=1036.659,-114.198,-77.055,168.139,37.792,157.088
C01367=1036.664,-113.949,-77.065,168.141,37.791,157.088
C01368=1036.670,-113.698,-77.073,168.144,37.791,157.087
C01369=1036.676,-113.448,-77.083,168.146,37.790,157.087
C01370=1036.682,-113.199,-77.093,168.149,37.789,157.087
C01371=1036.689,-112.949,-77.102,168.152,37.788,157.087
C01372=1036.694,-112.700,-77.111,168.155,37.787,157.087
C01373=1036.700,-112.450,-77.121,168.157,37.786,157.087
C01374=1036.707,-112.200,-77.130,168.160,37.785,157.087
C01375=1036.713,-111.950,-77.140,168.163,37.785,157.087
C01376=1036.719,-111.701,-77.150,168.166,37.784,157.087
C01377=1036.725,-111.450,-77.158,168.168,37.783,157.086
C01378=1036.730,-111.201,-77.168,168.170,37.782,157.086
C01379=1036.737,-110.951,-77.177,168.173,37.782,157.086
C01380=1036.743,-110.701,-77.187,168.175,37.781,157.086
C01381=1036.749,-110.452,-77.196,168.178,37.780,157.086
C01382=1036.755,-110.202,-77.206,168.181,37.779,157.086
C01383=1036.761,-109.952,-77.215,168.184,37.778,157.086
C01384=1036.767,-109.702,-77.225,168.186,37.777,157.086
C01385=1036.773,-109.453,-77.234,168.189,37.776,157.086
C01386=1036.779,-109.203,-77.244,168.192,37.776,157.086
C01387=1036.785,-108.953,-77.254,168.195,37.775,157.085
C01388=1036.791,-108.703,-77.263,168.197,37.774,157.085
C01389=1036.797,-108.454,-77.273,168.200,37.773,157.085
C01390=1036.803,-108.204,-77.283,168.202,37.773,157.085
C01391=1036.809,-107.954,-77.292,168.204,37.772,157.085
C01392=1036.815,-107.704,-77.302,168.207,37.771,157.085
C01393=1036.822,-107.454,-77.311,168.210,37.770,157.085
C01394=1036.828,-107.205,-77.321,168.213,37.770,157.085
C01395=1036.834,-106.955,-77.331,168.215,37.769,157.085
C01396=1036.840,-106.705,-77.341,168.218,37.768,157.085
C01397=1036.845,-106.456,-77.351,168.221,37.767,157.085
C01398=1036.851,-106.206,-77.360,168.223,37.767,157.084
C01399=1036.858,-105.957,-77.370,168.226,37.766,157.084
C01400=1036.864,-105.707,-77.379,168.229,37.765,157.084
C01401=1036.869,-105.457,-77.389,168.232,37.764,157.084
C01402=1036.875,-105.207,-77.399,168.234,37.764,157.084
C01403=1036.882,-104.958,-77.409,168.236,37.763,157.084
C01404=1036.888,-104.708,-77.419,168.239,37.762,157.084
C01405=1036.894,-104.458,-77.428,168.241,37.761,157.084
C01406=1036.900,-104.208,-77.439,168.244,37.761,157.084
C01407=1036.906,-103.958,-77.448,168.247,37.761,157.084
C01408=1036.912,-103.709,-77.458,168.249,37.760,157.084
C01409=1036.918,-103.459,-77.468,168.252,37.759,157.084
C01410=1036.924,-103.209,-77.478,168.255,37.758,157.083
C01411=1036.930,-102.959,-77.488,168.258,37.758,157.083
C01412=1036.937,-102.710,-77.498,168.260,37.757,157.083
C01413=1036.943,-102.460,-77.508,168.263,37.756,157.083
C01414=1036.948,-102.210,-77.518,168.266,37.755,157.083
C01415=1036.954,-101.961,-77.527,168.268,37.755,157.083
C01416=1036.961,-101.711,-77.538,168.271,37.754,157.083
C01417=1036.966,-101.461,-77.548,168.274,37.754,157.083
C01418=1036.972,-101.211,-77.557,168.275,37.753,157.083
C01419=1036.979,-100.962,-77.568,168.278,37.752,157.083
C01420=1036.985,-100.712,-77.577,168.281,37.751,157.083
C01421=1036.992,-100.425,-77.589,168.284,37.751,157.083
C01422=1036.999,-100.137,-77.600,168.287,37.750,157.083
C01423=1037.006,-99.850,-77.611,168.290,37.749,157.082
C01424=1037.013,-99.563,-77.624,168.293,37.748,157.082
C01425=1037.019,-99.313,-77.634,168.296,37.748,157.082
C01426=1037.025,-99.064,-77.643,168.298,37.747,157.082
C01427=1037.031,-98.814,-77.654,168.301,37.747,157.082
C01428=1037.037,-98.564,-77.664,168.304,37.746,157.082
C01429=1037.044,-98.315,-77.674,168.306,37.745,157.082
C01430=1037.049,-98.065,-77.684,168.309,37.745,157.082
///RCONF 1,0,0,0,0,0,0,0,0,0,0,0,0,0,0,0,0,0,0,0,0,0,0,0
C01431=1037.055,-97.815,-77.694,168.312,37.744,157.082
C01432=1037.062,-97.566,-77.704,168.314,37.743,157.082
C01433=1037.067,-97.316,-77.714,168.316,37.743,157.082
C01434=1037.074,-97.066,-77.725,168.319,37.742,157.082
C01435=1037.080,-96.816,-77.735,168.321,37.742,157.082
C01436=1037.086,-96.567,-77.745,168.324,37.741,157.082
C01437=1037.092,-96.317,-77.755,168.327,37.741,157.081
C01438=1037.098,-96.067,-77.766,168.329,37.740,157.081
C01439=1037.104,-95.817,-77.776,168.332,37.740,157.081
C01440=1037.109,-95.568,-77.787,168.335,37.739,157.081
C01441=1037.116,-95.318,-77.796,168.337,37.739,157.081
C01442=1037.121,-95.069,-77.807,168.340,37.738,157.081
C01443=1037.128,-94.818,-77.817,168.342,37.738,157.081
C01444=1037.134,-94.569,-77.828,168.345,37.737,157.081
C01445=1037.140,-94.319,-77.838,168.348,37.737,157.081
C01446=1037.146,-94.069,-77.848,168.350,37.736,157.081
C01447=1037.151,-93.820,-77.859,168.353,37.736,157.081
C01448=1037.158,-93.570,-77.869,168.356,37.735,157.081
C01449=1037.163,-93.321,-77.880,168.358,37.734,157.081
C01450=1037.170,-93.071,-77.890,168.361,37.734,157.081
C01451=1037.176,-92.821,-77.900,168.364,37.734,157.081
C01452=1037.182,-92.571,-77.911,168.366,37.734,157.081
C01453=1037.188,-92.322,-77.922,168.369,37.733,157.081
C01454=1037.194,-92.072,-77.932,168.370,37.732,157.081
C01455=1037.201,-91.822,-77.942,168.373,37.732,157.081
C01456=1037.206,-91.572,-77.953,168.376,37.731,157.081
C01457=1037.213,-91.323,-77.963,168.378,37.731,157.081
C01458=1037.218,-91.073,-77.974,168.381,37.730,157.080
C01459=1037.224,-90.824,-77.985,168.384,37.730,157.080
C01460=1037.231,-90.574,-77.995,168.386,37.730,157.080
C01461=1037.237,-90.324,-78.005,168.389,37.729,157.080
C01462=1037.243,-90.074,-78.016,168.391,37.729,157.080
C01463=1037.249,-89.825,-78.027,168.394,37.728,157.080
C01464=1037.255,-89.574,-78.037,168.397,37.727,157.080
C01465=1037.261,-89.325,-78.047,168.399,37.727,157.080
C01466=1037.267,-89.075,-78.058,168.402,37.726,157.080
C01467=1037.273,-88.826,-78.069,168.404,37.726,157.080
C01468=1037.280,-88.576,-78.080,168.407,37.726,157.080
C01469=1037.285,-88.326,-78.090,168.410,37.725,157.080
C01470=1037.292,-88.077,-78.100,168.412,37.725,157.080
C01471=1037.297,-87.827,-78.111,168.415,37.724,157.080
C01472=1037.305,-87.577,-78.122,168.418,37.724,157.080
C01473=1037.310,-87.328,-78.133,168.420,37.723,157.080
C01474=1037.316,-87.078,-78.143,168.423,37.723,157.080
C01475=1037.323,-86.828,-78.153,168.425,37.722,157.080
C01476=1037.329,-86.578,-78.164,168.428,37.722,157.080
C01477=1037.334,-86.329,-78.175,168.431,37.722,157.080
C01478=1037.341,-86.079,-78.186,168.432,37.721,157.079
C01479=1037.347,-85.830,-78.197,168.435,37.721,157.080
C01480=1037.354,-85.580,-78.207,168.437,37.720,157.079
C01481=1037.360,-85.330,-78.218,168.440,37.720,157.079
C01482=1037.365,-85.080,-78.228,168.443,37.719,157.079
C01483=1037.372,-84.831,-78.239,168.445,37.719,157.079
C01484=1037.378,-84.581,-78.250,168.448,37.718,157.079
C01485=1037.385,-84.296,-78.262,168.451,37.718,157.079
C01486=1037.393,-84.011,-78.275,168.454,37.717,157.079
C01487=1037.399,-83.727,-78.287,168.457,37.717,157.079
C01488=1037.407,-83.441,-78.299,168.460,37.717,157.079
C01489=1037.412,-83.192,-78.310,168.462,37.716,157.079
C01490=1037.419,-82.942,-78.321,168.465,37.716,157.079
C01491=1037.425,-82.693,-78.332,168.468,37.715,157.079
C01492=1037.431,-82.442,-78.343,168.470,37.715,157.079
C01493=1037.437,-82.193,-78.354,168.473,37.714,157.079
C01494=1037.444,-81.944,-78.364,168.475,37.714,157.079
C01495=1037.450,-81.693,-78.375,168.478,37.713,157.079
C01496=1037.456,-81.444,-78.386,168.481,37.713,157.079
C01497=1037.463,-81.194,-78.397,168.483,37.713,157.079
C01498=1037.469,-80.945,-78.408,168.486,37.712,157.079
C01499=1037.475,-80.694,-78.419,168.488,37.712,157.079
C01500=1037.481,-80.445,-78.429,168.491,37.711,157.079
C01501=1037.488,-80.195,-78.440,168.493,37.711,157.079
C01502=1037.493,-79.946,-78.451,168.496,37.710,157.079
C01503=1037.501,-79.696,-78.462,168.499,37.710,157.079
C01504=1037.506,-79.446,-78.473,168.501,37.710,157.079
C01505=1037.512,-79.197,-78.484,168.503,37.709,157.078
C01506=1037.519,-78.947,-78.496,168.506,37.709,157.078
C01507=1037.524,-78.698,-78.506,168.509,37.709,157.079
C01508=1037.531,-78.447,-78.518,168.510,37.708,157.078
C01509=1037.537,-78.198,-78.529,168.513,37.708,157.078
C01510=1037.543,-77.948,-78.540,168.515,37.708,157.078
C01511=1037.549,-77.699,-78.551,168.518,37.708,157.078
C01512=1037.555,-77.449,-78.563,168.521,37.707,157.078
C01513=1037.561,-77.199,-78.574,168.523,37.707,157.078
C01514=1037.567,-76.949,-78.585,168.526,37.707,157.078
C01515=1037.573,-76.700,-78.596,168.528,37.707,157.078
C01516=1037.580,-76.450,-78.607,168.531,37.706,157.078
C01517=1037.586,-76.201,-78.618,168.533,37.706,157.078
C01518=1037.593,-75.951,-78.629,168.536,37.706,157.078
C01519=1037.598,-75.701,-78.640,168.538,37.706,157.078
C01520=1037.605,-75.452,-78.652,168.541,37.706,157.078
C01521=1037.611,-75.202,-78.663,168.543,37.705,157.078
C01522=1037.617,-74.952,-78.674,168.546,37.705,157.078
C01523=1037.623,-74.703,-78.686,168.548,37.705,157.078
C01524=1037.629,-74.453,-78.697,168.551,37.704,157.078
C01525=1037.635,-74.203,-78.708,168.554,37.704,157.078
C01526=1037.642,-73.954,-78.720,168.556,37.704,157.078
C01527=1037.648,-73.704,-78.731,168.559,37.704,157.078
C01528=1037.654,-73.454,-78.742,168.561,37.704,157.078
C01529=1037.659,-73.205,-78.754,168.564,37.703,157.078
C01530=1037.665,-72.955,-78.765,168.566,37.703,157.078
C01531=1037.672,-72.705,-78.777,168.569,37.703,157.078
C01532=1037.678,-72.456,-78.788,168.571,37.703,157.078
C01533=1037.684,-72.205,-78.799,168.573,37.703,157.078
C01534=1037.690,-71.956,-78.812,168.576,37.702,157.078
C01535=1037.696,-71.706,-78.823,168.578,37.702,157.078
C01536=1037.702,-71.457,-78.834,168.581,37.702,157.078
C01537=1037.708,-71.207,-78.846,168.583,37.702,157.078
C01538=1037.714,-70.958,-78.857,168.586,37.701,157.078
C01539=1037.720,-70.708,-78.869,168.588,37.701,157.078
C01540=1037.726,-70.459,-78.881,168.591,37.701,157.078
C01541=1037.732,-70.209,-78.892,168.593,37.701,157.078
C01542=1037.739,-69.959,-78.904,168.596,37.701,157.078
C01543=1037.744,-69.709,-78.915,168.598,37.701,157.078
C01544=1037.751,-69.460,-78.927,168.601,37.701,157.078
C01545=1037.756,-69.210,-78.938,168.603,37.701,157.078
C01546=1037.763,-68.961,-78.950,168.606,37.701,157.078
C01547=1037.769,-68.710,-78.962,168.608,37.701,157.078
C01548=1037.775,-68.461,-78.974,168.611,37.701,157.078
C01549=1037.782,-68.178,-78.987,168.613,37.701,157.078
C01550=1037.789,-67.895,-79.000,168.616,37.700,157.078
C01551=1037.795,-67.612,-79.013,168.619,37.700,157.078
C01552=1037.802,-67.330,-79.027,168.622,37.700,157.078
C01553=1037.809,-67.080,-79.038,168.624,37.700,157.078
C01554=1037.815,-66.831,-79.050,168.627,37.700,157.078
C01555=1037.820,-66.581,-79.061,168.629,37.699,157.078
C01556=1037.827,-66.331,-79.073,168.632,37.699,157.078
C01557=1037.834,-66.082,-79.085,168.634,37.699,157.078
C01558=1037.840,-65.832,-79.096,168.637,37.699,157.078
C01559=1037.845,-65.582,-79.109,168.639,37.699,157.079
C01560=1037.852,-65.333,-79.121,168.642,37.699,157.079
C01561=1037.858,-65.083,-79.132,168.644,37.699,157.079
C01562=1037.864,-64.833,-79.144,168.647,37.699,157.079
C01563=1037.870,-64.584,-79.156,168.649,37.699,157.079
C01564=1037.877,-64.334,-79.167,168.651,37.699,157.079
C01565=1037.883,-64.085,-79.179,168.654,37.698,157.079
C01566=1037.889,-63.835,-79.191,168.656,37.698,157.079
C01567=1037.895,-63.585,-79.203,168.659,37.698,157.079
C01568=1037.902,-63.335,-79.215,168.661,37.698,157.079
C01569=1037.908,-63.086,-79.226,168.664,37.698,157.079
C01570=1037.914,-62.836,-79.239,168.666,37.698,157.079
C01571=1037.920,-62.587,-79.251,168.669,37.698,157.079
C01572=1037.927,-62.337,-79.262,168.671,37.698,157.079
C01573=1037.932,-62.087,-79.274,168.674,37.697,157.079
C01574=1037.939,-61.838,-79.286,168.676,37.697,157.079
C01575=1037.945,-61.588,-79.298,168.678,37.697,157.079
C01576=1037.952,-61.338,-79.309,168.681,37.697,157.079
C01577=1037.957,-61.089,-79.322,168.683,37.697,157.079
C01578=1037.963,-60.839,-79.333,168.686,37.697,157.079
C01579=1037.970,-60.590,-79.345,168.688,37.697,157.079
C01580=1037.976,-60.340,-79.358,168.691,37.697,157.079
C01581=1037.983,-60.090,-79.370,168.693,37.697,157.079
C01582=1037.988,-59.841,-79.381,168.696,37.697,157.079
C01583=1037.994,-59.591,-79.393,168.698,37.697,157.079
C01584=1038.001,-59.341,-79.405,168.700,37.697,157.079
C01585=1038.008,-59.092,-79.417,168.703,37.697,157.079
C01586=1038.014,-58.842,-79.430,168.705,37.696,157.079
C01587=1038.020,-58.592,-79.442,168.708,37.696,157.079
C01588=1038.026,-58.343,-79.453,168.710,37.696,157.079
C01589=1038.032,-58.094,-79.466,168.714,37.696,157.079
C01590=1038.039,-57.844,-79.478,168.716,37.696,157.079
C01591=1038.045,-57.594,-79.490,168.719,37.696,157.079
C01592=1038.051,-57.344,-79.502,168.721,37.696,157.079
C01593=1038.058,-57.094,-79.514,168.723,37.696,157.079
C01594=1038.064,-56.845,-79.526,168.726,37.696,157.079
C01595=1038.070,-56.595,-79.538,168.728,37.696,157.079
C01596=1038.076,-56.346,-79.550,168.731,37.696,157.079
C01597=1038.083,-56.096,-79.562,168.733,37.696,157.079
C01598=1038.089,-55.847,-79.574,168.736,37.696,157.079
C01599=1038.095,-55.597,-79.586,168.738,37.695,157.079
C01600=1038.102,-55.347,-79.598,168.740,37.695,157.079
C01601=1038.108,-55.098,-79.611,168.743,37.695,157.079
C01602=1038.115,-54.848,-79.623,168.745,37.695,157.079
C01603=1038.121,-54.598,-79.635,168.748,37.695,157.079
C01604=1038.127,-54.348,-79.647,168.750,37.695,157.079
C01605=1038.134,-54.099,-79.659,168.752,37.695,157.079
C01606=1038.141,-53.849,-79.671,168.755,37.695,157.079
C01607=1038.146,-53.599,-79.684,168.757,37.695,157.079
C01608=1038.153,-53.351,-79.696,168.760,37.695,157.079
C01609=1038.160,-53.101,-79.708,168.762,37.695,157.079
C01610=1038.166,-52.851,-79.721,168.765,37.695,157.079
C01611=1038.173,-52.601,-79.733,168.767,37.695,157.079
C01612=1038.178,-52.352,-79.745,168.769,37.695,157.079
C01613=1038.186,-52.071,-79.758,168.772,37.694,157.079
C01614=1038.193,-51.789,-79.773,168.775,37.694,157.079
C01615=1038.200,-51.507,-79.786,168.778,37.694,157.079
C01616=1038.207,-51.226,-79.801,168.780,37.694,157.079
C01617=1038.214,-50.976,-79.813,168.783,37.694,157.080
C01618=1038.221,-50.727,-79.825,168.785,37.694,157.080
C01619=1038.227,-50.477,-79.837,168.788,37.694,157.080
C01620=1038.233,-50.227,-79.850,168.790,37.694,157.080
C01621=1038.240,-49.978,-79.862,168.792,37.694,157.080
C01622=1038.245,-49.728,-79.875,168.795,37.694,157.080
C01623=1038.251,-49.478,-79.888,168.797,37.694,157.080
C01624=1038.258,-49.228,-79.900,168.799,37.694,157.080
C01625=1038.264,-48.979,-79.913,168.802,37.694,157.080
C01626=1038.270,-48.729,-79.925,168.804,37.695,157.080
C01627=1038.276,-48.479,-79.938,168.806,37.695,157.080
C01628=1038.283,-48.230,-79.951,168.809,37.695,157.080
C01629=1038.289,-47.981,-79.963,168.811,37.695,157.080
C01630=1038.295,-47.731,-79.976,168.813,37.695,157.080
C01631=1038.301,-47.481,-79.989,168.816,37.695,157.080
C01632=1038.308,-47.232,-80.001,168.818,37.695,157.080
C01633=1038.314,-46.982,-80.013,168.820,37.695,157.080
C01634=1038.320,-46.733,-80.027,168.823,37.695,157.080
C01635=1038.326,-46.483,-80.039,168.825,37.695,157.080
C01636=1038.332,-46.233,-80.051,168.827,37.695,157.080
C01637=1038.339,-45.984,-80.065,168.830,37.695,157.080
C01638=1038.344,-45.734,-80.077,168.832,37.696,157.080
C01639=1038.351,-45.485,-80.090,168.834,37.696,157.081
C01640=1038.357,-45.235,-80.102,168.837,37.696,157.081
C01641=1038.363,-44.985,-80.115,168.840,37.696,157.081
C01642=1038.369,-44.736,-80.128,168.842,37.696,157.081
C01643=1038.376,-44.487,-80.140,168.845,37.696,157.081
C01644=1038.382,-44.237,-80.153,168.847,37.696,157.081
C01645=1038.388,-43.987,-80.166,168.849,37.697,157.081
C01646=1038.394,-43.738,-80.179,168.852,37.697,157.081
C01647=1038.400,-43.488,-80.192,168.854,37.696,157.081
C01648=1038.408,-43.239,-80.205,168.856,37.696,157.081
C01649=1038.414,-42.989,-80.217,168.859,37.697,157.081
C01650=1038.420,-42.739,-80.230,168.861,37.697,157.081
C01651=1038.426,-42.490,-80.243,168.863,37.697,157.081
C01652=1038.433,-42.240,-80.255,168.866,37.697,157.081
C01653=1038.439,-41.991,-80.268,168.868,37.697,157.081
C01654=1038.445,-41.742,-80.282,168.870,37.697,157.081
C01655=1038.451,-41.492,-80.294,168.873,37.697,157.081
C01656=1038.458,-41.242,-80.307,168.875,37.698,157.081
C01657=1038.464,-40.992,-80.320,168.877,37.698,157.081
C01658=1038.471,-40.743,-80.333,168.880,37.698,157.081
C01659=1038.476,-40.493,-80.346,168.882,37.698,157.082
C01660=1038.483,-40.244,-80.359,168.884,37.698,157.082
C01661=1038.489,-39.994,-80.371,168.886,37.698,157.082
C01662=1038.496,-39.744,-80.384,168.889,37.698,157.082
C01663=1038.502,-39.495,-80.398,168.891,37.699,157.082
C01664=1038.508,-39.245,-80.410,168.893,37.698,157.082
C01665=1038.514,-38.996,-80.424,168.896,37.698,157.082
C01666=1038.521,-38.746,-80.436,168.898,37.699,157.082
C01667=1038.528,-38.496,-80.449,168.900,37.699,157.082
C01668=1038.533,-38.247,-80.463,168.904,37.699,157.082
C01669=1038.539,-37.997,-80.476,168.906,37.699,157.082
C01670=1038.546,-37.747,-80.489,168.908,37.699,157.082
C01671=1038.552,-37.498,-80.502,168.910,37.700,157.082
C01672=1038.559,-37.248,-80.516,168.913,37.700,157.082
C01673=1038.564,-36.998,-80.528,168.915,37.700,157.082
C01674=1038.571,-36.749,-80.542,168.917,37.700,157.082
C01675=1038.577,-36.500,-80.555,168.919,37.701,157.083
C01676=1038.583,-36.250,-80.567,168.922,37.701,157.083
C01677=1038.590,-35.969,-80.583,168.924,37.701,157.083
C01678=1038.597,-35.687,-80.598,168.927,37.701,157.083
C01679=1038.604,-35.407,-80.612,168.929,37.702,157.083
C01680=1038.612,-35.126,-80.627,168.932,37.702,157.083
C01681=1038.618,-34.877,-80.640,168.934,37.702,157.083
C01682=1038.625,-34.627,-80.654,168.936,37.702,157.083
C01683=1038.631,-34.377,-80.667,168.939,37.703,157.083
C01684=1038.636,-34.127,-80.680,168.941,37.703,157.083
C01685=1038.642,-33.878,-80.693,168.943,37.703,157.083
C01686=1038.649,-33.628,-80.707,168.945,37.703,157.083
C01687=1038.655,-33.379,-80.720,168.949,37.703,157.083
C01688=1038.661,-33.129,-80.734,168.951,37.704,157.083
C01689=1038.668,-32.879,-80.747,168.953,37.704,157.084
C01690=1038.674,-32.630,-80.760,168.955,37.704,157.084
C01691=1038.680,-32.380,-80.773,168.958,37.704,157.084
C01692=1038.687,-32.131,-80.786,168.960,37.705,157.084
C01693=1038.693,-31.881,-80.800,168.962,37.705,157.084
C01694=1038.700,-31.632,-80.813,168.964,37.705,157.084
C01695=1038.706,-31.383,-80.826,168.967,37.705,157.084
C01696=1038.713,-31.133,-80.840,168.969,37.706,157.084
C01697=1038.719,-30.883,-80.853,168.971,37.706,157.084
C01698=1038.725,-30.634,-80.867,168.973,37.706,157.084
C01699=1038.731,-30.384,-80.881,168.976,37.706,157.084
C01700=1038.737,-30.135,-80.894,168.978,37.706,157.084
C01701=1038.743,-29.885,-80.907,168.980,37.707,157.084
C01702=1038.750,-29.635,-80.920,168.982,37.707,157.084
C01703=1038.756,-29.385,-80.934,168.985,37.707,157.085
C01704=1038.762,-29.136,-80.947,168.987,37.707,157.085
C01705=1038.769,-28.886,-80.960,168.990,37.708,157.085
C01706=1038.775,-28.637,-80.974,168.992,37.708,157.085
C01707=1038.782,-28.388,-80.987,168.994,37.708,157.085
C01708=1038.789,-28.138,-81.001,168.997,37.708,157.085
C01709=1038.795,-27.888,-81.014,168.999,37.709,157.085
C01710=1038.801,-27.638,-81.028,169.001,37.709,157.085
C01711=1038.807,-27.389,-81.041,169.003,37.709,157.085
C01712=1038.813,-27.140,-81.055,169.006,37.709,157.085
C01713=1038.820,-26.890,-81.069,169.008,37.709,157.085
C01714=1038.827,-26.641,-81.082,169.010,37.710,157.085
C01715=1038.833,-26.391,-81.097,169.012,37.710,157.085
C01716=1038.839,-26.142,-81.110,169.014,37.710,157.086
C01717=1038.845,-25.892,-81.123,169.017,37.711,157.086
C01718=1038.851,-25.642,-81.137,169.019,37.711,157.086
C01719=1038.857,-25.393,-81.151,169.021,37.711,157.086
C01720=1038.864,-25.143,-81.164,169.023,37.712,157.086
C01721=1038.870,-24.894,-81.179,169.025,37.712,157.086
C01722=1038.876,-24.645,-81.192,169.028,37.712,157.086
C01723=1038.883,-24.395,-81.206,169.031,37.713,157.086
C01724=1038.888,-24.145,-81.220,169.033,37.713,157.086
C01725=1038.895,-23.895,-81.233,169.035,37.714,157.086
C01726=1038.901,-23.645,-81.247,169.037,37.714,157.087
C01727=1038.907,-23.397,-81.261,169.039,37.714,157.087
C01728=1038.914,-23.147,-81.275,169.042,37.715,157.087
C01729=1038.920,-22.897,-81.289,169.044,37.715,157.087
C01730=1038.926,-22.647,-81.302,169.046,37.715,157.087
C01731=1038.933,-22.399,-81.316,169.048,37.716,157.087
C01732=1038.939,-22.148,-81.330,169.050,37.716,157.087
C01733=1038.945,-21.899,-81.344,169.052,37.716,157.087
C01734=1038.951,-21.650,-81.357,169.055,37.717,157.087
C01735=1038.958,-21.400,-81.372,169.057,37.717,157.087
C01736=1038.964,-21.151,-81.385,169.059,37.717,157.087
C01737=1038.970,-20.901,-81.399,169.061,37.717,157.087
C01738=1038.977,-20.652,-81.413,169.064,37.718,157.088
C01739=1038.983,-20.402,-81.427,169.066,37.718,157.088
C01740=1038.989,-20.152,-81.441,169.069,37.718,157.088
C01741=1038.996,-19.871,-81.457,169.071,37.719,157.088
C01742=1039.004,-19.588,-81.472,169.074,37.720,157.088
C01743=1039.011,-19.307,-81.488,169.076,37.719,157.088
C01744=1039.018,-19.025,-81.504,169.078,37.720,157.088
C01745=1039.025,-18.775,-81.518,169.081,37.721,157.088
C01746=1039.030,-18.526,-81.532,169.083,37.721,157.088
C01747=1039.038,-18.276,-81.546,169.085,37.721,157.088
C01748=1039.044,-18.027,-81.559,169.087,37.722,157.089
C01749=1039.050,-17.777,-81.574,169.089,37.722,157.089
C01750=1039.056,-17.528,-81.588,169.091,37.722,157.089
C01751=1039.062,-17.278,-81.602,169.094,37.723,157.089
C01752=1039.069,-17.029,-81.616,169.097,37.723,157.089
C01753=1039.076,-16.779,-81.629,169.099,37.723,157.089
C01754=1039.082,-16.529,-81.644,169.101,37.723,157.089
C01755=1039.088,-16.280,-81.658,169.103,37.724,157.089
C01756=1039.094,-16.030,-81.672,169.105,37.724,157.089
C01757=1039.101,-15.781,-81.686,169.107,37.724,157.089
C01758=1039.107,-15.531,-81.700,169.110,37.725,157.089
C01759=1039.114,-15.283,-81.714,169.112,37.725,157.090
C01760=1039.120,-15.032,-81.728,169.114,37.725,157.090
C01761=1039.127,-14.783,-81.743,169.116,37.726,157.090
C01762=1039.132,-14.533,-81.757,169.118,37.727,157.090
C01763=1039.139,-14.284,-81.771,169.120,37.727,157.090
C01764=1039.145,-14.034,-81.785,169.122,37.727,157.090
C01765=1039.151,-13.785,-81.800,169.124,37.728,157.090
C01766=1039.158,-13.536,-81.814,169.127,37.728,157.090
C01767=1039.164,-13.286,-81.828,169.130,37.729,157.090
C01768=1039.170,-13.036,-81.843,169.132,37.729,157.091
C01769=1039.176,-12.787,-81.856,169.134,37.729,157.091
C01770=1039.183,-12.537,-81.871,169.136,37.730,157.091
C01771=1039.188,-12.288,-81.885,169.138,37.730,157.091
C01772=1039.195,-12.038,-81.899,169.140,37.731,157.091
C01773=1039.202,-11.789,-81.914,169.142,37.731,157.091
C01774=1039.207,-11.539,-81.928,169.144,37.732,157.091
C01775=1039.214,-11.290,-81.942,169.146,37.732,157.091
C01776=1039.220,-11.041,-81.957,169.148,37.733,157.091
C01777=1039.226,-10.791,-81.971,169.151,37.733,157.091
C01778=1039.233,-10.541,-81.986,169.154,37.733,157.092
C01779=1039.239,-10.292,-82.000,169.156,37.734,157.092
C01780=1039.245,-10.042,-82.014,169.158,37.734,157.092
C01781=1039.252,-9.793,-82.029,169.160,37.735,157.092
C01782=1039.258,-9.544,-82.043,169.162,37.735,157.092
C01783=1039.264,-9.293,-82.058,169.164,37.735,157.092
C01784=1039.271,-9.044,-82.072,169.166,37.736,157.092
C01785=1039.277,-8.795,-82.086,169.168,37.737,157.092
C01786=1039.283,-8.545,-82.101,169.170,37.737,157.092
C01787=1039.290,-8.295,-82.115,169.172,37.737,157.092
C01788=1039.296,-8.047,-82.130,169.175,37.738,157.093
C01789=1039.302,-7.797,-82.145,169.177,37.738,157.093
C01790=1039.309,-7.547,-82.160,169.179,37.738,157.093
C01791=1039.316,-7.297,-82.173,169.182,37.739,157.093
C01792=1039.321,-7.048,-82.188,169.184,37.739,157.093
C01793=1039.328,-6.799,-82.203,169.186,37.740,157.093
C01794=1039.335,-6.549,-82.217,169.188,37.740,157.093
C01795=1039.340,-6.300,-82.231,169.190,37.740,157.093
C01796=1039.347,-6.050,-82.246,169.192,37.741,157.093
C01797=1039.354,-5.801,-82.260,169.194,37.742,157.094
C01798=1039.360,-5.551,-82.275,169.196,37.742,157.094
C01799=1039.366,-5.302,-82.290,169.198,37.742,157.094
C01800=1039.373,-5.053,-82.304,169.201,37.743,157.094
C01801=1039.379,-4.802,-82.318,169.203,37.743,157.094
C01802=1039.386,-4.553,-82.333,169.206,37.744,157.094
C01803=1039.391,-4.304,-82.348,169.208,37.744,157.094
C01804=1039.399,-4.054,-82.362,169.210,37.744,157.094
C01805=1039.406,-3.771,-82.379,169.212,37.745,157.094
C01806=1039.413,-3.487,-82.395,169.215,37.745,157.095
C01807=1039.420,-3.204,-82.413,169.217,37.746,157.095
C01808=1039.427,-2.920,-82.429,169.219,37.747,157.095
C01809=1039.433,-2.671,-82.444,169.221,37.747,157.095
C01810=1039.439,-2.422,-82.459,169.223,37.748,157.095
C01811=1039.446,-2.172,-82.474,169.225,37.748,157.095
C01812=1039.452,-1.922,-82.489,169.227,37.749,157.095
